Yaskawa INFORM job: u_tourne2TRJ0.JBI

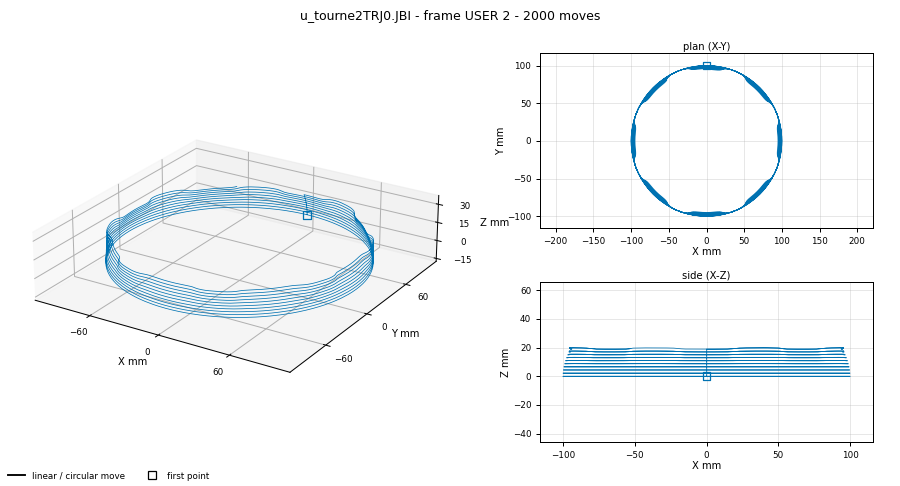
[picture p0: tool path of u_tourne2TRJ0.JBI in frame USER 2, 2000 of 2000 moves have a stored position in this frame; points joined in program order, loops and branches not executed]
/JOB
//NAME u_tourne2TRJ0
///FOLDERNAME DEMO
//POS
///NPOS 2000,0,0,0,0,0
///USER 2
///TOOL 7
///POSTYPE USER
///RECTAN
///RCONF 1,0,0,0,0,0,0,0,0,0,0,0,0,0,0,0,0,0,0,0,0,0,0,0
C00000=0.000,100.000,0.000,-180.0000,0.0000,0.0000
C00001=5.792,99.832,0.000,-180.0000,-0.0000,0.0000
C00002=10.988,99.394,0.000,-180.0000,-0.0000,0.0000
C00003=15.564,98.781,0.000,-180.0000,-0.0000,0.0000
C00004=18.698,98.237,0.000,-180.0000,-0.0000,0.0000
C00005=20.854,97.801,0.000,-180.0000,-0.0000,0.0000
C00006=22.593,97.414,0.000,-180.0000,-0.0000,0.0000
C00007=24.351,96.990,0.000,-180.0000,-0.0000,0.0000
C00008=26.550,96.411,0.000,-180.0000,-0.0000,0.0000
C00009=29.248,95.627,0.000,-180.0000,-0.0000,0.0000
C00010=32.094,94.710,0.000,-180.0000,-0.0000,0.0000
C00011=34.739,93.772,0.000,-180.0000,-0.0000,0.0000
C00012=37.121,92.855,0.000,-180.0000,-0.0000,0.0000
C00013=39.410,91.907,0.000,-180.0000,-0.0000,0.0000
C00014=41.743,90.871,0.000,-180.0000,-0.0000,0.0000
C00015=44.276,89.664,0.000,180.0000,0.0000,0.0000
C00016=46.937,88.300,0.000,180.0000,0.0000,0.0000
C00017=49.400,86.946,0.000,-180.0000,-0.0000,0.0000
C00018=51.363,85.801,0.000,-180.0000,-0.0000,0.0000
C00019=52.906,84.858,0.000,-180.0000,-0.0000,0.0000
C00020=54.410,83.902,0.000,-180.0000,-0.0000,0.0000
C00021=56.242,82.685,0.000,-180.0000,-0.0000,0.0000
C00022=58.844,80.854,0.000,-180.0000,-0.0000,0.0000
C00023=62.512,78.053,0.000,-180.0000,-0.0000,0.0000
C00024=66.496,74.687,0.000,-180.0000,-0.0000,0.0000
C00025=70.711,70.711,0.000,-180.0000,-0.0000,0.0000
C00026=74.687,66.496,0.000,-180.0000,-0.0000,0.0000
C00027=78.053,62.512,0.000,-180.0000,-0.0000,0.0000
C00028=80.854,58.844,0.000,180.0000,0.0000,0.0000
C00029=82.685,56.242,0.000,-180.0000,-0.0000,0.0000
C00030=83.902,54.410,0.000,-180.0000,-0.0000,0.0000
C00031=84.858,52.906,0.000,-180.0000,-0.0000,0.0000
C00032=85.801,51.363,0.000,-180.0000,-0.0000,0.0000
C00033=86.946,49.400,0.000,-180.0000,-0.0000,0.0000
C00034=88.300,46.937,0.000,-180.0000,-0.0000,0.0000
C00035=89.664,44.276,0.000,-180.0000,-0.0000,0.0000
C00036=90.871,41.743,0.000,-180.0000,-0.0000,0.0000
C00037=91.907,39.410,0.000,-180.0000,-0.0000,0.0000
C00038=92.855,37.121,0.000,-180.0000,-0.0000,0.0000
C00039=93.772,34.739,0.000,-180.0000,-0.0000,0.0000
C00040=94.710,32.094,0.000,-180.0000,-0.0000,0.0000
C00041=95.627,29.248,0.000,-180.0000,-0.0000,0.0000
C00042=96.411,26.550,0.000,-180.0000,-0.0000,0.0000
C00043=96.990,24.351,0.000,-180.0000,-0.0000,0.0000
C00044=97.414,22.593,0.000,-180.0000,-0.0000,0.0000
C00045=97.801,20.854,0.000,-180.0000,-0.0000,0.0000
C00046=98.237,18.698,0.000,-180.0000,-0.0000,0.0000
C00047=98.781,15.564,0.000,-180.0000,-0.0000,0.0000
C00048=99.394,10.988,0.000,-180.0000,-0.0000,0.0000
C00049=99.832,5.792,0.000,-180.0000,-0.0000,0.0000
C00050=100.000,0.000,0.000,-180.0000,-0.0000,0.0000
C00051=99.832,-5.792,0.000,180.0000,-0.0000,0.0000
C00052=99.394,-10.988,0.000,180.0000,-0.0000,0.0000
C00053=98.781,-15.564,0.000,180.0000,-0.0000,0.0000
C00054=98.237,-18.698,0.000,180.0000,-0.0000,0.0000
C00055=97.801,-20.854,0.000,180.0000,-0.0000,0.0000
C00056=97.414,-22.593,0.000,180.0000,-0.0000,0.0000
C00057=96.990,-24.351,0.000,180.0000,-0.0000,0.0000
C00058=96.411,-26.550,0.000,180.0000,-0.0000,0.0000
C00059=95.627,-29.248,0.000,180.0000,-0.0000,0.0000
C00060=94.710,-32.094,0.000,180.0000,-0.0000,0.0000
C00061=93.772,-34.739,0.000,180.0000,-0.0000,0.0000
C00062=92.855,-37.121,0.000,180.0000,-0.0000,0.0000
C00063=91.907,-39.410,0.000,180.0000,-0.0000,0.0000
C00064=90.871,-41.743,0.000,180.0000,-0.0000,0.0000
C00065=89.664,-44.276,0.000,180.0000,-0.0000,0.0000
C00066=88.300,-46.937,0.000,180.0000,-0.0000,0.0000
C00067=86.946,-49.400,0.000,180.0000,-0.0000,0.0000
C00068=85.801,-51.363,0.000,180.0000,-0.0000,0.0000
C00069=84.858,-52.906,0.000,180.0000,-0.0000,0.0000
C00070=83.902,-54.410,0.000,180.0000,-0.0000,0.0000
C00071=82.685,-56.242,0.000,180.0000,-0.0000,0.0000
C00072=80.854,-58.844,0.000,180.0000,-0.0000,0.0000
C00073=78.053,-62.512,0.000,180.0000,-0.0000,0.0000
C00074=74.687,-66.496,0.000,180.0000,-0.0000,0.0000
C00075=70.711,-70.711,0.000,180.0000,-0.0000,0.0000
C00076=66.496,-74.687,0.000,180.0000,-0.0000,0.0000
C00077=62.512,-78.053,0.000,180.0000,-0.0000,0.0000
C00078=58.844,-80.854,0.000,180.0000,-0.0000,0.0000
C00079=56.242,-82.685,0.000,180.0000,-0.0000,0.0000
C00080=54.410,-83.902,0.000,180.0000,-0.0000,0.0000
C00081=52.906,-84.858,0.000,180.0000,-0.0000,0.0000
C00082=51.363,-85.801,0.000,180.0000,-0.0000,0.0000
C00083=49.400,-86.946,0.000,-180.0000,0.0000,0.0000
C00084=46.937,-88.300,0.000,180.0000,-0.0000,0.0000
C00085=44.276,-89.664,0.000,180.0000,-0.0000,0.0000
C00086=41.743,-90.871,0.000,180.0000,-0.0000,0.0000
C00087=39.410,-91.907,0.000,180.0000,-0.0000,0.0000
C00088=37.121,-92.855,0.000,180.0000,-0.0000,0.0000
C00089=34.739,-93.772,0.000,180.0000,-0.0000,0.0000
C00090=32.094,-94.710,0.000,180.0000,-0.0000,0.0000
C00091=29.248,-95.627,0.000,180.0000,-0.0000,0.0000
C00092=26.550,-96.411,0.000,180.0000,-0.0000,0.0000
C00093=24.351,-96.990,0.000,180.0000,-0.0000,0.0000
C00094=22.593,-97.414,0.000,180.0000,-0.0000,0.0000
C00095=20.854,-97.801,0.000,180.0000,-0.0000,0.0000
C00096=18.698,-98.237,0.000,180.0000,-0.0000,0.0000
C00097=15.564,-98.781,0.000,180.0000,-0.0000,0.0000
C00098=10.988,-99.394,0.000,180.0000,-0.0000,0.0000
C00099=5.792,-99.832,0.000,180.0000,-0.0000,0.0000
C00100=0.000,-100.000,0.000,-180.0000,-0.0000,0.0000
C00101=0.000,-100.000,0.000,-180.0000,-0.0000,0.0000
C00102=-5.792,-99.832,0.000,-180.0000,-0.0000,0.0000
C00103=-10.988,-99.394,0.000,-180.0000,-0.0000,0.0000
C00104=-15.564,-98.781,0.000,-180.0000,-0.0000,0.0000
C00105=-18.698,-98.237,0.000,-180.0000,-0.0000,0.0000
C00106=-20.854,-97.801,0.000,-180.0000,-0.0000,0.0000
C00107=-22.593,-97.414,0.000,-180.0000,-0.0000,0.0000
C00108=-24.351,-96.990,0.000,-180.0000,-0.0000,0.0000
C00109=-26.550,-96.411,0.000,-180.0000,-0.0000,0.0000
C00110=-29.248,-95.627,0.000,-180.0000,-0.0000,0.0000
C00111=-32.094,-94.710,0.000,-180.0000,-0.0000,0.0000
C00112=-34.739,-93.772,0.000,-180.0000,-0.0000,0.0000
C00113=-37.121,-92.855,0.000,-180.0000,-0.0000,0.0000
C00114=-39.410,-91.907,0.000,-180.0000,-0.0000,0.0000
C00115=-41.743,-90.871,0.000,-180.0000,-0.0000,0.0000
C00116=-44.276,-89.664,0.000,-180.0000,-0.0000,0.0000
C00117=-46.937,-88.300,0.000,-180.0000,-0.0000,0.0000
C00118=-49.400,-86.946,0.000,-180.0000,-0.0000,0.0000
C00119=-51.363,-85.801,0.000,-180.0000,-0.0000,0.0000
C00120=-52.906,-84.858,0.000,-180.0000,-0.0000,0.0000
C00121=-54.410,-83.902,0.000,-180.0000,-0.0000,0.0000
C00122=-56.242,-82.685,0.000,-180.0000,-0.0000,0.0000
C00123=-58.844,-80.854,0.000,-180.0000,-0.0000,0.0000
C00124=-62.512,-78.053,0.000,-180.0000,-0.0000,0.0000
C00125=-66.496,-74.687,0.000,-180.0000,-0.0000,0.0000
C00126=-70.711,-70.711,0.000,-180.0000,-0.0000,0.0000
C00127=-74.687,-66.496,0.000,-180.0000,-0.0000,0.0000
C00128=-78.053,-62.512,0.000,-180.0000,-0.0000,0.0000
C00129=-80.854,-58.844,0.000,-180.0000,-0.0000,0.0000
C00130=-82.685,-56.242,0.000,-180.0000,-0.0000,0.0000
C00131=-83.902,-54.410,0.000,-180.0000,-0.0000,0.0000
C00132=-84.858,-52.906,0.000,-180.0000,-0.0000,0.0000
C00133=-85.801,-51.363,0.000,-180.0000,-0.0000,0.0000
C00134=-86.946,-49.400,0.000,-180.0000,-0.0000,0.0000
C00135=-88.300,-46.937,0.000,-180.0000,-0.0000,0.0000
C00136=-89.664,-44.276,0.000,-180.0000,-0.0000,0.0000
C00137=-90.871,-41.743,0.000,180.0000,0.0000,0.0000
C00138=-91.907,-39.410,0.000,180.0000,0.0000,0.0000
C00139=-92.855,-37.121,0.000,-180.0000,-0.0000,0.0000
C00140=-93.772,-34.739,0.000,-180.0000,-0.0000,0.0000
C00141=-94.710,-32.094,0.000,180.0000,0.0000,0.0000
C00142=-95.627,-29.248,0.000,180.0000,0.0000,0.0000
C00143=-96.411,-26.550,0.000,-180.0000,-0.0000,0.0000
C00144=-96.990,-24.351,0.000,-180.0000,-0.0000,0.0000
C00145=-97.414,-22.593,0.000,-180.0000,-0.0000,0.0000
C00146=-97.801,-20.854,0.000,-180.0000,-0.0000,0.0000
C00147=-98.237,-18.698,0.000,-180.0000,-0.0000,0.0000
C00148=-98.781,-15.564,0.000,-180.0000,-0.0000,0.0000
C00149=-99.394,-10.988,0.000,-180.0000,-0.0000,0.0000
C00150=-99.832,-5.792,0.000,-180.0000,-0.0000,0.0000
C00151=-100.000,0.000,0.000,180.0000,0.0000,0.0000
C00152=-99.832,5.792,0.000,-180.0000,0.0000,0.0000
C00153=-99.394,10.988,0.000,-180.0000,0.0000,0.0000
C00154=-98.781,15.564,0.000,-180.0000,0.0000,0.0000
C00155=-98.237,18.698,0.000,-180.0000,0.0000,0.0000
C00156=-97.801,20.854,0.000,-180.0000,0.0000,0.0000
C00157=-97.414,22.593,0.000,-180.0000,0.0000,0.0000
C00158=-96.990,24.351,0.000,-180.0000,0.0000,0.0000
C00159=-96.411,26.550,0.000,-180.0000,0.0000,0.0000
C00160=-95.627,29.248,0.000,-180.0000,0.0000,0.0000
C00161=-94.710,32.094,0.000,-180.0000,0.0000,0.0000
C00162=-93.772,34.739,0.000,-180.0000,0.0000,0.0000
C00163=-92.855,37.121,0.000,-180.0000,0.0000,0.0000
C00164=-91.907,39.410,0.000,-180.0000,0.0000,0.0000
C00165=-90.871,41.743,0.000,-180.0000,0.0000,0.0000
C00166=-89.664,44.276,0.000,-180.0000,0.0000,0.0000
C00167=-88.300,46.937,0.000,-180.0000,0.0000,0.0000
C00168=-86.946,49.400,0.000,-180.0000,0.0000,0.0000
C00169=-85.801,51.363,0.000,-180.0000,0.0000,0.0000
C00170=-84.858,52.906,0.000,-180.0000,0.0000,0.0000
C00171=-83.902,54.410,0.000,-180.0000,0.0000,0.0000
C00172=-82.685,56.242,0.000,-180.0000,0.0000,0.0000
C00173=-80.854,58.844,0.000,-180.0000,0.0000,0.0000
C00174=-78.053,62.512,0.000,-180.0000,0.0000,0.0000
C00175=-74.687,66.496,0.000,-180.0000,0.0000,0.0000
C00176=-70.711,70.711,0.000,-180.0000,0.0000,0.0000
C00177=-66.496,74.687,0.000,-180.0000,0.0000,0.0000
C00178=-62.512,78.053,0.000,-180.0000,0.0000,0.0000
C00179=-58.844,80.854,0.000,-180.0000,0.0000,0.0000
C00180=-56.242,82.685,0.000,-180.0000,0.0000,0.0000
C00181=-54.410,83.902,0.000,-180.0000,0.0000,0.0000
C00182=-52.906,84.858,0.000,-180.0000,0.0000,0.0000
C00183=-51.363,85.801,0.000,-180.0000,0.0000,0.0000
C00184=-49.400,86.946,0.000,-180.0000,0.0000,0.0000
C00185=-46.937,88.300,0.000,-180.0000,0.0000,0.0000
C00186=-44.276,89.664,0.000,-180.0000,0.0000,0.0000
C00187=-41.743,90.871,0.000,-180.0000,0.0000,0.0000
C00188=-39.410,91.907,0.000,-180.0000,0.0000,0.0000
C00189=-37.121,92.855,0.000,-180.0000,0.0000,0.0000
C00190=-34.739,93.772,0.000,-180.0000,0.0000,0.0000
C00191=-32.094,94.710,0.000,-180.0000,0.0000,0.0000
C00192=-29.248,95.627,0.000,-180.0000,0.0000,0.0000
C00193=-26.550,96.411,0.000,-180.0000,0.0000,0.0000
C00194=-24.351,96.990,0.000,-180.0000,0.0000,0.0000
C00195=-22.593,97.414,0.000,-180.0000,0.0000,0.0000
C00196=-20.854,97.801,0.000,-180.0000,0.0000,0.0000
C00197=-18.698,98.237,0.000,-180.0000,0.0000,0.0000
C00198=-15.564,98.781,0.000,-180.0000,0.0000,0.0000
C00199=-10.988,99.394,0.000,-180.0000,0.0000,0.0000
C00200=-5.792,99.832,0.000,-180.0000,0.0000,0.0000
C00201=0.000,100.000,0.000,-180.0000,0.0000,0.0000
C00202=0.000,99.921,2.199,-175.9401,0.0000,0.0000
C00203=5.785,99.754,2.199,-175.9458,-0.2355,0.0000
C00204=10.976,99.317,2.199,-175.9687,-0.4480,0.0000
C00205=15.549,98.707,2.199,-176.1467,-0.6030,0.0000
C00206=18.681,98.171,2.199,-176.5598,-0.6429,0.0000
C00207=20.835,97.748,2.199,-177.1510,-0.5909,0.0000
C00208=22.573,97.375,2.200,-177.8335,-0.4817,0.0000
C00209=24.330,96.965,2.200,-178.5158,-0.3611,0.0000
C00210=26.527,96.399,2.200,-179.1062,-0.2407,0.0000
C00211=29.226,95.625,2.200,-179.5703,-0.1318,0.0000
C00212=32.077,94.713,2.200,-179.8797,-0.0401,0.0000
C00213=34.728,93.776,2.200,-179.9828,-0.0057,0.0000
C00214=37.118,92.856,2.200,-180.0000,-0.0000,0.0000
C00215=39.413,91.905,2.200,-180.0000,-0.0000,0.0000
C00216=41.753,90.866,2.200,-179.9828,-0.0115,0.0000
C00217=44.291,89.654,2.200,-179.8854,-0.0573,0.0000
C00218=46.951,88.283,2.200,-179.6047,-0.2120,0.0000
C00219=49.407,86.922,2.200,-179.1978,-0.4641,0.0000
C00220=51.360,85.768,2.200,-178.6934,-0.7909,0.0000
C00221=52.893,84.816,2.200,-178.1256,-1.1925,0.0000
C00222=54.385,83.851,2.199,-177.5690,-1.6002,0.0000
C00223=56.208,82.627,2.199,-177.1150,-1.9797,0.0000
C00224=58.802,80.791,2.199,-176.8504,-2.3016,0.0000
C00225=62.466,77.989,2.199,-176.8326,-2.5372,0.0000
C00226=66.446,74.627,2.199,-176.9643,-2.7034,0.0000
C00227=70.655,70.655,2.199,-177.1247,-2.8753,0.0000
C00228=74.627,66.446,2.199,-177.2966,-3.0357,0.0000
C00229=77.989,62.466,2.199,-177.4628,-3.1674,0.0000
C00230=80.791,58.802,2.199,-177.6984,-3.1496,0.0000
C00231=82.627,56.208,2.199,-178.0203,-2.8850,0.0000
C00232=83.851,54.385,2.199,-178.3998,-2.4310,0.0000
C00233=84.816,52.893,2.200,-178.8075,-1.8744,0.0000
C00234=85.768,51.360,2.200,-179.2091,-1.3066,0.0000
C00235=86.922,49.407,2.200,-179.5359,-0.8022,0.0000
C00236=88.283,46.951,2.200,-179.7880,-0.3953,0.0000
C00237=89.654,44.291,2.200,-179.9427,-0.1146,0.0000
C00238=90.866,41.753,2.200,-179.9885,-0.0172,0.0000
C00239=91.905,39.413,2.200,-180.0000,-0.0000,0.0000
C00240=92.856,37.118,2.200,-180.0000,-0.0000,0.0000
C00241=93.776,34.728,2.200,-179.9943,-0.0172,0.0000
C00242=94.713,32.077,2.200,-179.9599,-0.1203,0.0000
C00243=95.625,29.226,2.200,-179.8682,-0.4297,0.0000
C00244=96.399,26.527,2.200,-179.7593,-0.8938,0.0000
C00245=96.965,24.330,2.200,-179.6389,-1.4842,0.0000
C00246=97.375,22.573,2.200,-179.5183,-2.1665,0.0000
C00247=97.748,20.835,2.199,-179.4091,-2.8490,0.0000
C00248=98.171,18.681,2.199,-179.3571,-3.4402,0.0000
C00249=98.707,15.549,2.199,-179.3970,-3.8533,0.0000
C00250=99.317,10.976,2.199,-179.5520,-4.0313,0.0000
C00251=99.754,5.785,2.199,-179.7645,-4.0542,0.0000
C00252=99.921,0.000,2.199,180.0000,-4.0599,0.0000
C00253=99.754,-5.785,2.199,179.7645,-4.0542,0.0000
C00254=99.317,-10.976,2.199,179.5520,-4.0313,0.0000
C00255=98.707,-15.549,2.199,179.3970,-3.8533,0.0000
C00256=98.171,-18.681,2.199,179.3571,-3.4402,0.0000
C00257=97.748,-20.835,2.199,179.4091,-2.8490,0.0000
C00258=97.375,-22.573,2.200,179.5183,-2.1665,0.0000
C00259=96.965,-24.330,2.200,179.6389,-1.4842,0.0000
C00260=96.399,-26.527,2.200,179.7593,-0.8938,0.0000
C00261=95.625,-29.226,2.200,179.8682,-0.4297,0.0000
C00262=94.713,-32.077,2.200,179.9599,-0.1203,0.0000
C00263=93.776,-34.728,2.200,179.9943,-0.0172,0.0000
C00264=92.856,-37.118,2.200,180.0000,-0.0000,0.0000
C00265=91.905,-39.413,2.200,180.0000,-0.0000,0.0000
C00266=90.866,-41.753,2.200,179.9885,-0.0172,0.0000
C00267=89.654,-44.291,2.200,179.9427,-0.1146,0.0000
C00268=88.283,-46.951,2.200,179.7880,-0.3953,0.0000
C00269=86.922,-49.407,2.200,179.5359,-0.8022,0.0000
C00270=85.768,-51.360,2.200,179.2091,-1.3066,0.0000
C00271=84.816,-52.893,2.200,178.8075,-1.8744,0.0000
C00272=83.851,-54.385,2.199,178.3998,-2.4310,0.0000
C00273=82.627,-56.208,2.199,178.0203,-2.8850,0.0000
C00274=80.791,-58.802,2.199,177.6984,-3.1496,0.0000
C00275=77.989,-62.466,2.199,177.4628,-3.1674,0.0000
C00276=74.627,-66.446,2.199,177.2966,-3.0357,0.0000
C00277=70.655,-70.655,2.199,177.1247,-2.8753,0.0000
C00278=66.446,-74.627,2.199,176.9643,-2.7034,0.0000
C00279=62.466,-77.989,2.199,176.8326,-2.5372,0.0000
C00280=58.802,-80.791,2.199,176.8504,-2.3016,0.0000
C00281=56.208,-82.627,2.199,177.1150,-1.9797,0.0000
C00282=54.385,-83.851,2.199,177.5690,-1.6002,0.0000
C00283=52.893,-84.816,2.200,178.1256,-1.1925,0.0000
C00284=51.360,-85.768,2.200,178.6934,-0.7909,0.0000
C00285=49.407,-86.922,2.200,179.1978,-0.4641,0.0000
C00286=46.951,-88.283,2.200,179.6047,-0.2120,0.0000
C00287=44.291,-89.654,2.200,179.8854,-0.0573,0.0000
C00288=41.753,-90.866,2.200,179.9828,-0.0115,0.0000
C00289=39.413,-91.905,2.200,180.0000,-0.0000,0.0000
C00290=37.118,-92.856,2.200,180.0000,-0.0000,0.0000
C00291=34.728,-93.776,2.200,179.9828,-0.0057,0.0000
C00292=32.077,-94.713,2.200,179.8797,-0.0401,0.0000
C00293=29.226,-95.625,2.200,179.5703,-0.1318,0.0000
C00294=26.527,-96.399,2.200,179.1062,-0.2407,0.0000
C00295=24.330,-96.965,2.200,178.5158,-0.3611,0.0000
C00296=22.573,-97.375,2.200,177.8335,-0.4817,0.0000
C00297=20.835,-97.748,2.199,177.1510,-0.5909,0.0000
C00298=18.681,-98.171,2.199,176.5598,-0.6429,0.0000
C00299=15.549,-98.707,2.199,176.1467,-0.6030,0.0000
C00300=10.976,-99.317,2.199,175.9687,-0.4480,0.0000
C00301=5.785,-99.754,2.199,175.9458,-0.2355,0.0000
C00302=0.000,-99.921,2.199,175.9401,0.0000,0.0000
C00303=0.000,-99.921,2.199,175.9401,0.0000,0.0000
C00304=-5.785,-99.754,2.199,175.9458,0.2355,0.0000
C00305=-10.976,-99.317,2.199,175.9687,0.4480,0.0000
C00306=-15.549,-98.707,2.199,176.1467,0.6030,0.0000
C00307=-18.681,-98.171,2.199,176.5598,0.6429,0.0000
C00308=-20.835,-97.748,2.199,177.1510,0.5909,0.0000
C00309=-22.573,-97.375,2.200,177.8335,0.4817,0.0000
C00310=-24.330,-96.965,2.200,178.5158,0.3611,0.0000
C00311=-26.527,-96.399,2.200,179.1062,0.2407,0.0000
C00312=-29.226,-95.625,2.200,179.5703,0.1318,0.0000
C00313=-32.077,-94.713,2.200,179.8797,0.0401,0.0000
C00314=-34.728,-93.776,2.200,179.9828,0.0057,0.0000
C00315=-37.118,-92.856,2.200,180.0000,0.0000,0.0000
C00316=-39.413,-91.905,2.200,180.0000,0.0000,0.0000
C00317=-41.753,-90.866,2.200,179.9828,0.0115,0.0000
C00318=-44.291,-89.654,2.200,179.8854,0.0573,0.0000
C00319=-46.951,-88.283,2.200,179.6047,0.2120,0.0000
C00320=-49.407,-86.922,2.200,179.1978,0.4641,0.0000
C00321=-51.360,-85.768,2.200,178.6934,0.7909,0.0000
C00322=-52.893,-84.816,2.200,178.1256,1.1925,0.0000
C00323=-54.385,-83.851,2.199,177.5690,1.6002,0.0000
C00324=-56.208,-82.627,2.199,177.1150,1.9797,0.0000
C00325=-58.802,-80.791,2.199,176.8504,2.3016,0.0000
C00326=-62.466,-77.989,2.199,176.8326,2.5372,0.0000
C00327=-66.446,-74.627,2.199,176.9643,2.7034,0.0000
C00328=-70.655,-70.655,2.199,177.1247,2.8753,0.0000
C00329=-74.627,-66.446,2.199,177.2966,3.0357,0.0000
C00330=-77.989,-62.466,2.199,177.4628,3.1674,0.0000
C00331=-80.791,-58.802,2.199,177.6984,3.1496,0.0000
C00332=-82.627,-56.208,2.199,178.0203,2.8850,0.0000
C00333=-83.851,-54.385,2.199,178.3998,2.4310,0.0000
C00334=-84.816,-52.893,2.200,178.8075,1.8744,0.0000
C00335=-85.768,-51.360,2.200,179.2091,1.3066,0.0000
C00336=-86.922,-49.407,2.200,179.5359,0.8022,0.0000
C00337=-88.283,-46.951,2.200,179.7880,0.3953,0.0000
C00338=-89.654,-44.291,2.200,179.9427,0.1146,0.0000
C00339=-90.866,-41.753,2.200,179.9885,0.0172,0.0000
C00340=-91.905,-39.413,2.200,180.0000,0.0000,0.0000
C00341=-92.856,-37.118,2.200,180.0000,0.0000,0.0000
C00342=-93.776,-34.728,2.200,179.9943,0.0172,0.0000
C00343=-94.713,-32.077,2.200,179.9599,0.1203,0.0000
C00344=-95.625,-29.226,2.200,179.8682,0.4297,0.0000
C00345=-96.399,-26.527,2.200,179.7593,0.8938,0.0000
C00346=-96.965,-24.330,2.200,179.6389,1.4842,0.0000
C00347=-97.375,-22.573,2.200,179.5183,2.1665,0.0000
C00348=-97.748,-20.835,2.199,179.4091,2.8490,0.0000
C00349=-98.171,-18.681,2.199,179.3571,3.4402,0.0000
C00350=-98.707,-15.549,2.199,179.3970,3.8533,0.0000
C00351=-99.317,-10.976,2.199,179.5520,4.0313,0.0000
C00352=-99.754,-5.785,2.199,179.7645,4.0542,0.0000
C00353=-99.921,0.000,2.199,-180.0000,4.0599,0.0000
C00354=-99.754,5.785,2.199,-179.7645,4.0542,0.0000
C00355=-99.317,10.976,2.199,-179.5520,4.0313,0.0000
C00356=-98.707,15.549,2.199,-179.3970,3.8533,0.0000
C00357=-98.171,18.681,2.199,-179.3571,3.4402,0.0000
C00358=-97.748,20.835,2.199,-179.4091,2.8490,0.0000
C00359=-97.375,22.573,2.200,-179.5183,2.1665,0.0000
C00360=-96.965,24.330,2.200,-179.6389,1.4842,0.0000
C00361=-96.399,26.527,2.200,-179.7593,0.8938,0.0000
C00362=-95.625,29.226,2.200,-179.8682,0.4297,0.0000
C00363=-94.713,32.077,2.200,-179.9599,0.1203,0.0000
C00364=-93.776,34.728,2.200,-179.9943,0.0172,0.0000
C00365=-92.856,37.118,2.200,-180.0000,0.0000,0.0000
C00366=-91.905,39.413,2.200,-180.0000,0.0000,0.0000
C00367=-90.866,41.753,2.200,-179.9885,0.0172,0.0000
C00368=-89.654,44.291,2.200,-179.9427,0.1146,0.0000
C00369=-88.283,46.951,2.200,-179.7880,0.3953,0.0000
C00370=-86.922,49.407,2.200,-179.5359,0.8022,0.0000
C00371=-85.768,51.360,2.200,-179.2091,1.3066,0.0000
C00372=-84.816,52.893,2.200,-178.8075,1.8744,0.0000
C00373=-83.851,54.385,2.199,-178.3998,2.4310,0.0000
C00374=-82.627,56.208,2.199,-178.0203,2.8850,0.0000
C00375=-80.791,58.802,2.199,-177.6984,3.1496,0.0000
C00376=-77.989,62.466,2.199,-177.4628,3.1674,0.0000
C00377=-74.627,66.446,2.199,-177.2966,3.0357,0.0000
C00378=-70.655,70.655,2.199,-177.1247,2.8753,0.0000
C00379=-66.446,74.627,2.199,-176.9643,2.7034,0.0000
C00380=-62.466,77.989,2.199,-176.8326,2.5372,0.0000
C00381=-58.802,80.791,2.199,-176.8504,2.3016,0.0000
C00382=-56.208,82.627,2.199,-177.1150,1.9797,0.0000
C00383=-54.385,83.851,2.199,-177.5690,1.6002,0.0000
C00384=-52.893,84.816,2.200,-178.1256,1.1925,0.0000
C00385=-51.360,85.768,2.200,-178.6934,0.7909,0.0000
C00386=-49.407,86.922,2.200,-179.1978,0.4641,0.0000
C00387=-46.951,88.283,2.200,-179.6047,0.2120,0.0000
C00388=-44.291,89.654,2.200,-179.8854,0.0573,0.0000
C00389=-41.753,90.866,2.200,-179.9828,0.0115,0.0000
C00390=-39.413,91.905,2.200,-180.0000,0.0000,0.0000
C00391=-37.118,92.856,2.200,-180.0000,0.0000,0.0000
C00392=-34.728,93.776,2.200,-179.9828,0.0057,0.0000
C00393=-32.077,94.713,2.200,-179.8797,0.0401,0.0000
C00394=-29.226,95.625,2.200,-179.5703,0.1318,0.0000
C00395=-26.527,96.399,2.200,-179.1062,0.2407,0.0000
C00396=-24.330,96.965,2.200,-178.5158,0.3611,0.0000
C00397=-22.573,97.375,2.200,-177.8335,0.4817,0.0000
C00398=-20.835,97.748,2.199,-177.1510,0.5909,0.0000
C00399=-18.681,98.171,2.199,-176.5598,0.6429,0.0000
C00400=-15.549,98.707,2.199,-176.1467,0.6030,0.0000
C00401=-10.976,99.317,2.199,-175.9687,0.4480,0.0000
C00402=-5.785,99.754,2.199,-175.9458,0.2355,0.0000
C00403=0.000,99.921,2.199,-175.9401,0.0000,0.0000
C00404=0.000,99.691,4.387,-172.1025,0.0000,0.0000
C00405=5.764,99.524,4.387,-172.1138,-0.4628,0.0000
C00406=10.941,99.090,4.387,-172.1592,-0.8618,0.0000
C00407=15.506,98.490,4.388,-172.4997,-1.1444,0.0000
C00408=18.630,97.979,4.390,-173.2915,-1.1769,0.0000
C00409=20.779,97.591,4.393,-174.4382,-1.0363,0.0000
C00410=22.514,97.259,4.396,-175.7731,-0.8388,0.0000
C00411=24.268,96.890,4.398,-177.1167,-0.6425,0.0000
C00412=26.460,96.362,4.399,-178.2693,-0.4471,0.0000
C00413=29.164,95.617,4.399,-179.1806,-0.2407,0.0000
C00414=32.027,94.722,4.399,-179.7708,-0.0745,0.0000
C00415=34.697,93.786,4.400,-179.9656,-0.0115,0.0000
C00416=37.107,92.860,4.400,-179.9943,-0.0000,0.0000
C00417=39.424,91.901,4.400,-179.9943,-0.0000,0.0000
C00418=41.782,90.851,4.400,-179.9656,-0.0172,0.0000
C00419=44.332,89.625,4.399,-179.7823,-0.1089,0.0000
C00420=46.990,88.233,4.399,-179.2494,-0.4126,0.0000
C00421=49.428,86.848,4.399,-178.4583,-0.9114,0.0000
C00422=51.352,85.672,4.398,-177.5060,-1.5830,0.0000
C00423=52.853,84.692,4.396,-176.4194,-2.4003,0.0000
C00424=54.314,83.700,4.393,-175.3293,-3.2095,0.0000
C00425=56.108,82.455,4.390,-174.4208,-3.9289,0.0000
C00426=58.679,80.608,4.388,-173.8788,-4.5167,0.0000
C00427=62.331,77.804,4.387,-173.8345,-4.9565,0.0000
C00428=66.299,74.450,4.387,-174.0804,-5.2721,0.0000
C00429=70.493,70.493,4.387,-174.3954,-5.6046,0.0000
C00430=74.450,66.299,4.387,-174.7279,-5.9196,0.0000
C00431=77.804,62.331,4.387,-175.0435,-6.1655,0.0000
C00432=80.608,58.679,4.388,-175.4833,-6.1212,0.0000
C00433=82.455,56.108,4.390,-176.0711,-5.5792,0.0000
C00434=83.700,54.314,4.393,-176.7905,-4.6707,0.0000
C00435=84.692,52.853,4.396,-177.5997,-3.5806,0.0000
C00436=85.672,51.352,4.398,-178.4170,-2.4940,0.0000
C00437=86.848,49.428,4.399,-179.0886,-1.5417,0.0000
C00438=88.233,46.990,4.399,-179.5874,-0.7506,0.0000
C00439=89.625,44.332,4.399,-179.8911,-0.2177,0.0000
C00440=90.851,41.782,4.400,-179.9828,-0.0344,0.0000
C00441=91.901,39.424,4.400,-180.0000,-0.0057,0.0000
C00442=92.860,37.107,4.400,-180.0000,-0.0057,0.0000
C00443=93.786,34.697,4.400,-179.9885,-0.0344,0.0000
C00444=94.722,32.027,4.399,-179.9255,-0.2292,0.0000
C00445=95.617,29.164,4.399,-179.7593,-0.8194,0.0000
C00446=96.362,26.460,4.399,-179.5529,-1.7307,0.0000
C00447=96.890,24.268,4.398,-179.3575,-2.8833,0.0000
C00448=97.259,22.514,4.396,-179.1612,-4.2269,0.0000
C00449=97.591,20.779,4.393,-178.9637,-5.5618,0.0000
C00450=97.979,18.630,4.390,-178.8231,-6.7085,0.0000
C00451=98.490,15.506,4.388,-178.8556,-7.5003,0.0000
C00452=99.090,10.941,4.387,-179.1382,-7.8408,0.0000
C00453=99.524,5.764,4.387,-179.5372,-7.8862,0.0000
C00454=99.691,0.000,4.387,180.0000,-7.8975,0.0000
C00455=99.524,-5.764,4.387,179.5372,-7.8862,0.0000
C00456=99.090,-10.941,4.387,179.1382,-7.8408,0.0000
C00457=98.490,-15.506,4.388,178.8556,-7.5003,0.0000
C00458=97.979,-18.630,4.390,178.8231,-6.7085,0.0000
C00459=97.591,-20.779,4.393,178.9637,-5.5618,0.0000
C00460=97.259,-22.514,4.396,179.1612,-4.2269,0.0000
C00461=96.890,-24.268,4.398,179.3575,-2.8833,0.0000
C00462=96.362,-26.460,4.399,179.5529,-1.7307,0.0000
C00463=95.617,-29.164,4.399,179.7593,-0.8194,0.0000
C00464=94.722,-32.027,4.399,179.9255,-0.2292,0.0000
C00465=93.786,-34.697,4.400,179.9885,-0.0344,0.0000
C00466=92.860,-37.107,4.400,180.0000,-0.0057,0.0000
C00467=91.901,-39.424,4.400,180.0000,-0.0057,0.0000
C00468=90.851,-41.782,4.400,179.9828,-0.0344,0.0000
C00469=89.625,-44.332,4.399,179.8911,-0.2177,0.0000
C00470=88.233,-46.990,4.399,179.5874,-0.7506,0.0000
C00471=86.848,-49.428,4.399,179.0886,-1.5417,0.0000
C00472=85.672,-51.352,4.398,178.4170,-2.4940,0.0000
C00473=84.692,-52.853,4.396,177.5997,-3.5806,0.0000
C00474=83.700,-54.314,4.393,176.7905,-4.6707,0.0000
C00475=82.455,-56.108,4.390,176.0711,-5.5792,0.0000
C00476=80.608,-58.679,4.388,175.4833,-6.1212,0.0000
C00477=77.804,-62.331,4.387,175.0435,-6.1655,0.0000
C00478=74.450,-66.299,4.387,174.7279,-5.9196,0.0000
C00479=70.493,-70.493,4.387,174.3954,-5.6046,0.0000
C00480=66.299,-74.450,4.387,174.0804,-5.2721,0.0000
C00481=62.331,-77.804,4.387,173.8345,-4.9565,0.0000
C00482=58.679,-80.608,4.388,173.8788,-4.5167,0.0000
C00483=56.108,-82.455,4.390,174.4208,-3.9289,0.0000
C00484=54.314,-83.700,4.393,175.3293,-3.2095,0.0000
C00485=52.853,-84.692,4.396,176.4194,-2.4003,0.0000
C00486=51.352,-85.672,4.398,177.5060,-1.5830,0.0000
C00487=49.428,-86.848,4.399,178.4583,-0.9114,0.0000
C00488=46.990,-88.233,4.399,179.2494,-0.4126,0.0000
C00489=44.332,-89.625,4.399,179.7823,-0.1089,0.0000
C00490=41.782,-90.851,4.400,179.9656,-0.0172,0.0000
C00491=39.424,-91.901,4.400,179.9943,-0.0000,0.0000
C00492=37.107,-92.860,4.400,179.9943,-0.0000,0.0000
C00493=34.697,-93.786,4.400,179.9656,-0.0115,0.0000
C00494=32.027,-94.722,4.399,179.7708,-0.0745,0.0000
C00495=29.164,-95.617,4.399,179.1806,-0.2407,0.0000
C00496=26.460,-96.362,4.399,178.2693,-0.4471,0.0000
C00497=24.268,-96.890,4.398,177.1167,-0.6425,0.0000
C00498=22.514,-97.259,4.396,175.7731,-0.8388,0.0000
C00499=20.779,-97.591,4.393,174.4382,-1.0363,0.0000
C00500=18.630,-97.979,4.390,173.2915,-1.1769,0.0000
C00501=15.506,-98.490,4.388,172.4997,-1.1444,0.0000
C00502=10.941,-99.090,4.387,172.1592,-0.8618,0.0000
C00503=5.764,-99.524,4.387,172.1138,-0.4628,0.0000
C00504=0.000,-99.691,4.387,172.1025,0.0000,0.0000
C00505=0.000,-99.691,4.387,172.1025,0.0000,0.0000
C00506=-5.764,-99.524,4.387,172.1138,0.4628,0.0000
C00507=-10.941,-99.090,4.387,172.1592,0.8618,0.0000
C00508=-15.506,-98.490,4.388,172.4997,1.1444,0.0000
C00509=-18.630,-97.979,4.390,173.2915,1.1769,0.0000
C00510=-20.779,-97.591,4.393,174.4382,1.0363,0.0000
C00511=-22.514,-97.259,4.396,175.7731,0.8388,0.0000
C00512=-24.268,-96.890,4.398,177.1167,0.6425,0.0000
C00513=-26.460,-96.362,4.399,178.2693,0.4471,0.0000
C00514=-29.164,-95.617,4.399,179.1806,0.2407,0.0000
C00515=-32.027,-94.722,4.399,179.7708,0.0745,0.0000
C00516=-34.697,-93.786,4.400,179.9656,0.0115,0.0000
C00517=-37.107,-92.860,4.400,179.9943,0.0000,0.0000
C00518=-39.424,-91.901,4.400,179.9943,0.0000,0.0000
C00519=-41.782,-90.851,4.400,179.9656,0.0172,0.0000
C00520=-44.332,-89.625,4.399,179.7823,0.1089,0.0000
C00521=-46.990,-88.233,4.399,179.2494,0.4126,0.0000
C00522=-49.428,-86.848,4.399,178.4583,0.9114,0.0000
C00523=-51.352,-85.672,4.398,177.5060,1.5830,0.0000
C00524=-52.853,-84.692,4.396,176.4194,2.4003,0.0000
C00525=-54.314,-83.700,4.393,175.3293,3.2095,0.0000
C00526=-56.108,-82.455,4.390,174.4208,3.9289,0.0000
C00527=-58.679,-80.608,4.388,173.8788,4.5167,0.0000
C00528=-62.331,-77.804,4.387,173.8345,4.9565,0.0000
C00529=-66.299,-74.450,4.387,174.0804,5.2721,0.0000
C00530=-70.493,-70.493,4.387,174.3954,5.6046,0.0000
C00531=-74.450,-66.299,4.387,174.7279,5.9196,0.0000
C00532=-77.804,-62.331,4.387,175.0435,6.1655,0.0000
C00533=-80.608,-58.679,4.388,175.4833,6.1212,0.0000
C00534=-82.455,-56.108,4.390,176.0711,5.5792,0.0000
C00535=-83.700,-54.314,4.393,176.7905,4.6707,0.0000
C00536=-84.692,-52.853,4.396,177.5997,3.5806,0.0000
C00537=-85.672,-51.352,4.398,178.4170,2.4940,0.0000
C00538=-86.848,-49.428,4.399,179.0886,1.5417,0.0000
C00539=-88.233,-46.990,4.399,179.5874,0.7506,0.0000
C00540=-89.625,-44.332,4.399,179.8911,0.2177,0.0000
C00541=-90.851,-41.782,4.400,179.9828,0.0344,0.0000
C00542=-91.901,-39.424,4.400,180.0000,0.0057,0.0000
C00543=-92.860,-37.107,4.400,180.0000,0.0057,0.0000
C00544=-93.786,-34.697,4.400,179.9885,0.0344,0.0000
C00545=-94.722,-32.027,4.399,179.9255,0.2292,0.0000
C00546=-95.617,-29.164,4.399,179.7593,0.8194,0.0000
C00547=-96.362,-26.460,4.399,179.5529,1.7307,0.0000
C00548=-96.890,-24.268,4.398,179.3575,2.8833,0.0000
C00549=-97.259,-22.514,4.396,179.1612,4.2269,0.0000
C00550=-97.591,-20.779,4.393,178.9637,5.5618,0.0000
C00551=-97.979,-18.630,4.390,178.8231,6.7085,0.0000
C00552=-98.490,-15.506,4.388,178.8556,7.5003,0.0000
C00553=-99.090,-10.941,4.387,179.1382,7.8408,0.0000
C00554=-99.524,-5.764,4.387,179.5372,7.8862,0.0000
C00555=-99.691,0.000,4.387,-180.0000,7.8975,0.0000
C00556=-99.524,5.764,4.387,-179.5372,7.8862,0.0000
C00557=-99.090,10.941,4.387,-179.1382,7.8408,0.0000
C00558=-98.490,15.506,4.388,-178.8556,7.5003,0.0000
C00559=-97.979,18.630,4.390,-178.8231,6.7085,0.0000
C00560=-97.591,20.779,4.393,-178.9637,5.5618,0.0000
C00561=-97.259,22.514,4.396,-179.1612,4.2269,0.0000
C00562=-96.890,24.268,4.398,-179.3575,2.8833,0.0000
C00563=-96.362,26.460,4.399,-179.5529,1.7307,0.0000
C00564=-95.617,29.164,4.399,-179.7593,0.8194,0.0000
C00565=-94.722,32.027,4.399,-179.9255,0.2292,0.0000
C00566=-93.786,34.697,4.400,-179.9885,0.0344,0.0000
C00567=-92.860,37.107,4.400,-180.0000,0.0057,0.0000
C00568=-91.901,39.424,4.400,-180.0000,0.0057,0.0000
C00569=-90.851,41.782,4.400,-179.9828,0.0344,0.0000
C00570=-89.625,44.332,4.399,-179.8911,0.2177,0.0000
C00571=-88.233,46.990,4.399,-179.5874,0.7506,0.0000
C00572=-86.848,49.428,4.399,-179.0886,1.5417,0.0000
C00573=-85.672,51.352,4.398,-178.4170,2.4940,0.0000
C00574=-84.692,52.853,4.396,-177.5997,3.5806,0.0000
C00575=-83.700,54.314,4.393,-176.7905,4.6707,0.0000
C00576=-82.455,56.108,4.390,-176.0711,5.5792,0.0000
C00577=-80.608,58.679,4.388,-175.4833,6.1212,0.0000
C00578=-77.804,62.331,4.387,-175.0435,6.1655,0.0000
C00579=-74.450,66.299,4.387,-174.7279,5.9196,0.0000
C00580=-70.493,70.493,4.387,-174.3954,5.6046,0.0000
C00581=-66.299,74.450,4.387,-174.0804,5.2721,0.0000
C00582=-62.331,77.804,4.387,-173.8345,4.9565,0.0000
C00583=-58.679,80.608,4.388,-173.8788,4.5167,0.0000
C00584=-56.108,82.455,4.390,-174.4208,3.9289,0.0000
C00585=-54.314,83.700,4.393,-175.3293,3.2095,0.0000
C00586=-52.853,84.692,4.396,-176.4194,2.4003,0.0000
C00587=-51.352,85.672,4.398,-177.5060,1.5830,0.0000
C00588=-49.428,86.848,4.399,-178.4583,0.9114,0.0000
C00589=-46.990,88.233,4.399,-179.2494,0.4126,0.0000
C00590=-44.332,89.625,4.399,-179.7823,0.1089,0.0000
C00591=-41.782,90.851,4.400,-179.9656,0.0172,0.0000
C00592=-39.424,91.901,4.400,-179.9943,0.0000,0.0000
C00593=-37.107,92.860,4.400,-179.9943,0.0000,0.0000
C00594=-34.697,93.786,4.400,-179.9656,0.0115,0.0000
C00595=-32.027,94.722,4.399,-179.7708,0.0745,0.0000
C00596=-29.164,95.617,4.399,-179.1806,0.2407,0.0000
C00597=-26.460,96.362,4.399,-178.2693,0.4471,0.0000
C00598=-24.268,96.890,4.398,-177.1167,0.6425,0.0000
C00599=-22.514,97.259,4.396,-175.7731,0.8388,0.0000
C00600=-20.779,97.591,4.393,-174.4382,1.0363,0.0000
C00601=-18.630,97.979,4.390,-173.2915,1.1769,0.0000
C00602=-15.506,98.490,4.388,-172.4997,1.1444,0.0000
C00603=-10.941,99.090,4.387,-172.1592,0.8618,0.0000
C00604=-5.764,99.524,4.387,-172.1138,0.4628,0.0000
C00605=0.000,99.691,4.387,-172.1025,0.0000,0.0000
C00606=0.000,99.321,6.555,-168.5271,0.0000,0.0000
C00607=5.730,99.155,6.555,-168.5440,-0.6723,0.0000
C00608=10.884,98.723,6.555,-168.6125,-1.2508,0.0000
C00609=15.437,98.140,6.558,-169.0891,-1.6049,0.0000
C00610=18.547,97.668,6.566,-170.2258,-1.5293,0.0000
C00611=20.687,97.336,6.576,-171.8926,-1.2386,0.0000
C00612=22.417,97.071,6.585,-173.8623,-0.9682,0.0000
C00613=24.167,96.770,6.592,-175.8307,-0.7870,0.0000
C00614=26.351,96.303,6.595,-177.5124,-0.5850,0.0000
C00615=29.062,95.605,6.597,-178.8311,-0.3266,0.0000
C00616=31.947,94.737,6.598,-179.6791,-0.1031,0.0000
C00617=34.646,93.803,6.599,-179.9484,-0.0172,0.0000
C00618=37.090,92.867,6.600,-179.9943,-0.0000,0.0000
C00619=39.440,91.893,6.600,-179.9943,-0.0000,0.0000
C00620=41.830,90.827,6.599,-179.9484,-0.0229,0.0000
C00621=44.399,89.579,6.598,-179.7021,-0.1547,0.0000
C00622=47.053,88.152,6.597,-178.9457,-0.5960,0.0000
C00623=49.464,86.729,6.595,-177.8216,-1.3476,0.0000
C00624=51.338,85.515,6.592,-176.4941,-2.3943,0.0000
C00625=52.788,84.491,6.585,-174.9698,-3.6664,0.0000
C00626=54.199,83.455,6.576,-173.3785,-4.8853,0.0000
C00627=55.947,82.176,6.566,-171.9913,-5.8770,0.0000
C00628=58.480,80.311,6.558,-171.1284,-6.6482,0.0000
C00629=62.112,77.504,6.555,-171.0304,-7.2336,0.0000
C00630=66.061,74.165,6.555,-171.3778,-7.6884,0.0000
C00631=70.230,70.230,6.555,-171.8355,-8.1645,0.0000
C00632=74.165,66.061,6.555,-172.3116,-8.6222,0.0000
C00633=77.504,62.112,6.555,-172.7664,-8.9696,0.0000
C00634=80.311,58.480,6.558,-173.3518,-8.8716,0.0000
C00635=82.176,55.947,6.566,-174.1230,-8.0087,0.0000
C00636=83.455,54.199,6.576,-175.1147,-6.6215,0.0000
C00637=84.491,52.788,6.585,-176.3336,-5.0302,0.0000
C00638=85.515,51.338,6.592,-177.6057,-3.5059,0.0000
C00639=86.729,49.464,6.595,-178.6524,-2.1784,0.0000
C00640=88.152,47.053,6.597,-179.4040,-1.0543,0.0000
C00641=89.579,44.399,6.598,-179.8453,-0.2979,0.0000
C00642=90.827,41.830,6.599,-179.9771,-0.0516,0.0000
C00643=91.893,39.440,6.600,-180.0000,-0.0057,0.0000
C00644=92.867,37.090,6.600,-180.0000,-0.0057,0.0000
C00645=93.803,34.646,6.599,-179.9828,-0.0516,0.0000
C00646=94.737,31.947,6.598,-179.8969,-0.3209,0.0000
C00647=95.605,29.062,6.597,-179.6734,-1.1689,0.0000
C00648=96.303,26.351,6.595,-179.4150,-2.4876,0.0000
C00649=96.770,24.167,6.592,-179.2130,-4.1693,0.0000
C00650=97.071,22.417,6.585,-179.0318,-6.1377,0.0000
C00651=97.336,20.687,6.576,-178.7614,-8.1074,0.0000
C00652=97.668,18.547,6.566,-178.4707,-9.7742,0.0000
C00653=98.140,15.437,6.558,-178.3951,-10.9109,0.0000
C00654=98.723,10.884,6.555,-178.7492,-11.3875,0.0000
C00655=99.155,5.730,6.555,-179.3277,-11.4560,0.0000
C00656=99.321,0.000,6.555,180.0000,-11.4729,0.0000
C00657=99.155,-5.730,6.555,179.3277,-11.4560,0.0000
C00658=98.723,-10.884,6.555,178.7492,-11.3875,0.0000
C00659=98.140,-15.437,6.558,178.3951,-10.9109,0.0000
C00660=97.668,-18.547,6.566,178.4707,-9.7742,0.0000
C00661=97.336,-20.687,6.576,178.7614,-8.1074,0.0000
C00662=97.071,-22.417,6.585,179.0318,-6.1377,0.0000
C00663=96.770,-24.167,6.592,179.2130,-4.1693,0.0000
C00664=96.303,-26.351,6.595,179.4150,-2.4876,0.0000
C00665=95.605,-29.062,6.597,179.6734,-1.1689,0.0000
C00666=94.737,-31.947,6.598,179.8969,-0.3209,0.0000
C00667=93.803,-34.646,6.599,179.9828,-0.0516,0.0000
C00668=92.867,-37.090,6.600,180.0000,-0.0057,0.0000
C00669=91.893,-39.440,6.600,180.0000,-0.0057,0.0000
C00670=90.827,-41.830,6.599,179.9771,-0.0516,0.0000
C00671=89.579,-44.399,6.598,179.8453,-0.2979,0.0000
C00672=88.152,-47.053,6.597,179.4040,-1.0543,0.0000
C00673=86.729,-49.464,6.595,178.6524,-2.1784,0.0000
C00674=85.515,-51.338,6.592,177.6057,-3.5059,0.0000
C00675=84.491,-52.788,6.585,176.3336,-5.0302,0.0000
C00676=83.455,-54.199,6.576,175.1147,-6.6215,0.0000
C00677=82.176,-55.947,6.566,174.1230,-8.0087,0.0000
C00678=80.311,-58.480,6.558,173.3518,-8.8716,0.0000
C00679=77.504,-62.112,6.555,172.7664,-8.9696,0.0000
C00680=74.165,-66.061,6.555,172.3116,-8.6222,0.0000
C00681=70.230,-70.230,6.555,171.8355,-8.1645,0.0000
C00682=66.061,-74.165,6.555,171.3778,-7.6884,0.0000
C00683=62.112,-77.504,6.555,171.0304,-7.2336,0.0000
C00684=58.480,-80.311,6.558,171.1284,-6.6482,0.0000
C00685=55.947,-82.176,6.566,171.9913,-5.8770,0.0000
C00686=54.199,-83.455,6.576,173.3785,-4.8853,0.0000
C00687=52.788,-84.491,6.585,174.9698,-3.6664,0.0000
C00688=51.338,-85.515,6.592,176.4941,-2.3943,0.0000
C00689=49.464,-86.729,6.595,177.8216,-1.3476,0.0000
C00690=47.053,-88.152,6.597,178.9457,-0.5960,0.0000
C00691=44.399,-89.579,6.598,179.7021,-0.1547,0.0000
C00692=41.830,-90.827,6.599,179.9484,-0.0229,0.0000
C00693=39.440,-91.893,6.600,179.9943,-0.0000,0.0000
C00694=37.090,-92.867,6.600,179.9943,-0.0000,0.0000
C00695=34.646,-93.803,6.599,179.9484,-0.0172,0.0000
C00696=31.947,-94.737,6.598,179.6791,-0.1031,0.0000
C00697=29.062,-95.605,6.597,178.8311,-0.3266,0.0000
C00698=26.351,-96.303,6.595,177.5124,-0.5850,0.0000
C00699=24.167,-96.770,6.592,175.8307,-0.7870,0.0000
C00700=22.417,-97.071,6.585,173.8623,-0.9682,0.0000
C00701=20.687,-97.336,6.576,171.8926,-1.2386,0.0000
C00702=18.547,-97.668,6.566,170.2258,-1.5293,0.0000
C00703=15.437,-98.140,6.558,169.0891,-1.6049,0.0000
C00704=10.884,-98.723,6.555,168.6125,-1.2508,0.0000
C00705=5.730,-99.155,6.555,168.5440,-0.6723,0.0000
C00706=0.000,-99.321,6.555,168.5271,0.0000,0.0000
C00707=0.000,-99.321,6.555,168.5271,0.0000,0.0000
C00708=-5.730,-99.155,6.555,168.5440,0.6723,0.0000
C00709=-10.884,-98.723,6.555,168.6125,1.2508,0.0000
C00710=-15.437,-98.140,6.558,169.0891,1.6049,0.0000
C00711=-18.547,-97.668,6.566,170.2258,1.5293,0.0000
C00712=-20.687,-97.336,6.576,171.8926,1.2386,0.0000
C00713=-22.417,-97.071,6.585,173.8623,0.9682,0.0000
C00714=-24.167,-96.770,6.592,175.8307,0.7870,0.0000
C00715=-26.351,-96.303,6.595,177.5124,0.5850,0.0000
C00716=-29.062,-95.605,6.597,178.8311,0.3266,0.0000
C00717=-31.947,-94.737,6.598,179.6791,0.1031,0.0000
C00718=-34.646,-93.803,6.599,179.9484,0.0172,0.0000
C00719=-37.090,-92.867,6.600,179.9943,0.0000,0.0000
C00720=-39.440,-91.893,6.600,179.9943,0.0000,0.0000
C00721=-41.830,-90.827,6.599,179.9484,0.0229,0.0000
C00722=-44.399,-89.579,6.598,179.7021,0.1547,0.0000
C00723=-47.053,-88.152,6.597,178.9457,0.5960,0.0000
C00724=-49.464,-86.729,6.595,177.8216,1.3476,0.0000
C00725=-51.338,-85.515,6.592,176.4941,2.3943,0.0000
C00726=-52.788,-84.491,6.585,174.9698,3.6664,0.0000
C00727=-54.199,-83.455,6.576,173.3785,4.8853,0.0000
C00728=-55.947,-82.176,6.566,171.9913,5.8770,0.0000
C00729=-58.480,-80.311,6.558,171.1284,6.6482,0.0000
C00730=-62.112,-77.504,6.555,171.0304,7.2336,0.0000
C00731=-66.061,-74.165,6.555,171.3778,7.6884,0.0000
C00732=-70.230,-70.230,6.555,171.8355,8.1645,0.0000
C00733=-74.165,-66.061,6.555,172.3116,8.6222,0.0000
C00734=-77.504,-62.112,6.555,172.7664,8.9696,0.0000
C00735=-80.311,-58.480,6.558,173.3518,8.8716,0.0000
C00736=-82.176,-55.947,6.566,174.1230,8.0087,0.0000
C00737=-83.455,-54.199,6.576,175.1147,6.6215,0.0000
C00738=-84.491,-52.788,6.585,176.3336,5.0302,0.0000
C00739=-85.515,-51.338,6.592,177.6057,3.5059,0.0000
C00740=-86.729,-49.464,6.595,178.6524,2.1784,0.0000
C00741=-88.152,-47.053,6.597,179.4040,1.0543,0.0000
C00742=-89.579,-44.399,6.598,179.8453,0.2979,0.0000
C00743=-90.827,-41.830,6.599,179.9771,0.0516,0.0000
C00744=-91.893,-39.440,6.600,180.0000,0.0057,0.0000
C00745=-92.867,-37.090,6.600,180.0000,0.0057,0.0000
C00746=-93.803,-34.646,6.599,179.9828,0.0516,0.0000
C00747=-94.737,-31.947,6.598,179.8969,0.3209,0.0000
C00748=-95.605,-29.062,6.597,179.6734,1.1689,0.0000
C00749=-96.303,-26.351,6.595,179.4150,2.4876,0.0000
C00750=-96.770,-24.167,6.592,179.2130,4.1693,0.0000
C00751=-97.071,-22.417,6.585,179.0318,6.1377,0.0000
C00752=-97.336,-20.687,6.576,178.7614,8.1074,0.0000
C00753=-97.668,-18.547,6.566,178.4707,9.7742,0.0000
C00754=-98.140,-15.437,6.558,178.3951,10.9109,0.0000
C00755=-98.723,-10.884,6.555,178.7492,11.3875,0.0000
C00756=-99.155,-5.730,6.555,179.3277,11.4560,0.0000
C00757=-99.321,0.000,6.555,-180.0000,11.4729,0.0000
C00758=-99.155,5.730,6.555,-179.3277,11.4560,0.0000
C00759=-98.723,10.884,6.555,-178.7492,11.3875,0.0000
C00760=-98.140,15.437,6.558,-178.3951,10.9109,0.0000
C00761=-97.668,18.547,6.566,-178.4707,9.7742,0.0000
C00762=-97.336,20.687,6.576,-178.7614,8.1074,0.0000
C00763=-97.071,22.417,6.585,-179.0318,6.1377,0.0000
C00764=-96.770,24.167,6.592,-179.2130,4.1693,0.0000
C00765=-96.303,26.351,6.595,-179.4150,2.4876,0.0000
C00766=-95.605,29.062,6.597,-179.6734,1.1689,0.0000
C00767=-94.737,31.947,6.598,-179.8969,0.3209,0.0000
C00768=-93.803,34.646,6.599,-179.9828,0.0516,0.0000
C00769=-92.867,37.090,6.600,-180.0000,0.0057,0.0000
C00770=-91.893,39.440,6.600,-180.0000,0.0057,0.0000
C00771=-90.827,41.830,6.599,-179.9771,0.0516,0.0000
C00772=-89.579,44.399,6.598,-179.8453,0.2979,0.0000
C00773=-88.152,47.053,6.597,-179.4040,1.0543,0.0000
C00774=-86.729,49.464,6.595,-178.6524,2.1784,0.0000
C00775=-85.515,51.338,6.592,-177.6057,3.5059,0.0000
C00776=-84.491,52.788,6.585,-176.3336,5.0302,0.0000
C00777=-83.455,54.199,6.576,-175.1147,6.6215,0.0000
C00778=-82.176,55.947,6.566,-174.1230,8.0087,0.0000
C00779=-80.311,58.480,6.558,-173.3518,8.8716,0.0000
C00780=-77.504,62.112,6.555,-172.7664,8.9696,0.0000
C00781=-74.165,66.061,6.555,-172.3116,8.6222,0.0000
C00782=-70.230,70.230,6.555,-171.8355,8.1645,0.0000
C00783=-66.061,74.165,6.555,-171.3778,7.6884,0.0000
C00784=-62.112,77.504,6.555,-171.0304,7.2336,0.0000
C00785=-58.480,80.311,6.558,-171.1284,6.6482,0.0000
C00786=-55.947,82.176,6.566,-171.9913,5.8770,0.0000
C00787=-54.199,83.455,6.576,-173.3785,4.8853,0.0000
C00788=-52.788,84.491,6.585,-174.9698,3.6664,0.0000
C00789=-51.338,85.515,6.592,-176.4941,2.3943,0.0000
C00790=-49.464,86.729,6.595,-177.8216,1.3476,0.0000
C00791=-47.053,88.152,6.597,-178.9457,0.5960,0.0000
C00792=-44.399,89.579,6.598,-179.7021,0.1547,0.0000
C00793=-41.830,90.827,6.599,-179.9484,0.0229,0.0000
C00794=-39.440,91.893,6.600,-179.9943,0.0000,0.0000
C00795=-37.090,92.867,6.600,-179.9943,0.0000,0.0000
C00796=-34.646,93.803,6.599,-179.9484,0.0172,0.0000
C00797=-31.947,94.737,6.598,-179.6791,0.1031,0.0000
C00798=-29.062,95.605,6.597,-178.8311,0.3266,0.0000
C00799=-26.351,96.303,6.595,-177.5124,0.5850,0.0000
C00800=-24.167,96.770,6.592,-175.8307,0.7870,0.0000
C00801=-22.417,97.071,6.585,-173.8623,0.9682,0.0000
C00802=-20.687,97.336,6.576,-171.8926,1.2386,0.0000
C00803=-18.547,97.668,6.566,-170.2258,1.5293,0.0000
C00804=-15.437,98.140,6.558,-169.0891,1.6049,0.0000
C00805=-10.884,98.723,6.555,-168.6125,1.2508,0.0000
C00806=-5.730,99.155,6.555,-168.5440,0.6723,0.0000
C00807=0.000,99.321,6.555,-168.5271,0.0000,0.0000
C00808=0.000,98.820,8.697,-165.2384,0.0000,0.0000
C00809=5.684,98.656,8.697,-165.2550,-0.8768,0.0000
C00810=10.807,98.229,8.698,-165.3451,-1.6051,0.0000
C00811=15.344,97.668,8.705,-165.9346,-1.9495,0.0000
C00812=18.436,97.247,8.723,-167.3804,-1.6441,0.0000
C00813=20.563,96.991,8.745,-169.5521,-1.1187,0.0000
C00814=22.286,96.814,8.767,-172.1365,-0.8040,0.0000
C00815=24.029,96.606,8.782,-174.6920,-0.7538,0.0000
C00816=26.202,96.222,8.789,-176.8469,-0.6485,0.0000
C00817=28.922,95.588,8.792,-178.5388,-0.3783,0.0000
C00818=31.837,94.757,8.795,-179.6161,-0.1203,0.0000
C00819=34.577,93.826,8.798,-179.9370,-0.0229,0.0000
C00820=37.066,92.876,8.800,-179.9943,-0.0057,0.0000
C00821=39.463,91.883,8.800,-179.9943,-0.0057,0.0000
C00822=41.895,90.794,8.798,-179.9370,-0.0286,0.0000
C00823=44.491,89.515,8.795,-179.6448,-0.1891,0.0000
C00824=47.140,88.042,8.792,-178.6992,-0.7622,0.0000
C00825=49.511,86.567,8.789,-177.3105,-1.7727,0.0000
C00826=51.320,85.302,8.782,-175.7091,-3.2251,0.0000
C00827=52.699,84.217,8.767,-173.8631,-5.0139,0.0000
C00828=54.043,83.124,8.745,-171.7932,-6.6483,0.0000
C00829=55.728,81.800,8.723,-169.8751,-7.8561,0.0000
C00830=58.212,79.911,8.705,-168.6219,-8.7026,0.0000
C00831=61.817,77.101,8.698,-168.4294,-9.3768,0.0000
C00832=65.741,73.780,8.697,-168.8611,-9.9421,0.0000
C00833=69.877,69.877,8.697,-169.4440,-10.5560,0.0000
C00834=73.780,65.741,8.697,-170.0579,-11.1389,0.0000
C00835=77.101,61.817,8.698,-170.6232,-11.5706,0.0000
C00836=79.911,58.212,8.705,-171.2974,-11.3781,0.0000
C00837=81.800,55.728,8.723,-172.1439,-10.1249,0.0000
C00838=83.124,54.043,8.745,-173.3517,-8.2068,0.0000
C00839=84.217,52.699,8.767,-174.9861,-6.1369,0.0000
C00840=85.302,51.320,8.782,-176.7749,-4.2909,0.0000
C00841=86.567,49.511,8.789,-178.2273,-2.6895,0.0000
C00842=88.042,47.140,8.792,-179.2378,-1.3008,0.0000
C00843=89.515,44.491,8.795,-179.8109,-0.3552,0.0000
C00844=90.794,41.895,8.798,-179.9714,-0.0630,0.0000
C00845=91.883,39.463,8.800,-179.9943,-0.0057,0.0000
C00846=92.876,37.066,8.800,-179.9943,-0.0057,0.0000
C00847=93.826,34.577,8.798,-179.9771,-0.0630,0.0000
C00848=94.757,31.837,8.795,-179.8797,-0.3839,0.0000
C00849=95.588,28.922,8.792,-179.6217,-1.4612,0.0000
C00850=96.222,26.202,8.789,-179.3515,-3.1531,0.0000
C00851=96.606,24.029,8.782,-179.2462,-5.3080,0.0000
C00852=96.814,22.286,8.767,-179.1960,-7.8635,0.0000
C00853=96.991,20.563,8.745,-178.8813,-10.4479,0.0000
C00854=97.247,18.436,8.723,-178.3559,-12.6196,0.0000
C00855=97.668,15.344,8.705,-178.0505,-14.0654,0.0000
C00856=98.229,10.807,8.698,-178.3949,-14.6549,0.0000
C00857=98.656,5.684,8.697,-179.1232,-14.7450,0.0000
C00858=98.820,0.000,8.697,180.0000,-14.7616,0.0000
C00859=98.656,-5.684,8.697,179.1232,-14.7450,0.0000
C00860=98.229,-10.807,8.698,178.3949,-14.6549,0.0000
C00861=97.668,-15.344,8.705,178.0505,-14.0654,0.0000
C00862=97.247,-18.436,8.723,178.3559,-12.6196,0.0000
C00863=96.991,-20.563,8.745,178.8813,-10.4479,0.0000
C00864=96.814,-22.286,8.767,179.1960,-7.8635,0.0000
C00865=96.606,-24.029,8.782,179.2462,-5.3080,0.0000
C00866=96.222,-26.202,8.789,179.3515,-3.1531,0.0000
C00867=95.588,-28.922,8.792,179.6217,-1.4612,0.0000
C00868=94.757,-31.837,8.795,179.8797,-0.3839,0.0000
C00869=93.826,-34.577,8.798,179.9771,-0.0630,0.0000
C00870=92.876,-37.066,8.800,179.9943,-0.0057,0.0000
C00871=91.883,-39.463,8.800,179.9943,-0.0057,0.0000
C00872=90.794,-41.895,8.798,179.9714,-0.0630,0.0000
C00873=89.515,-44.491,8.795,179.8109,-0.3552,0.0000
C00874=88.042,-47.140,8.792,179.2378,-1.3008,0.0000
C00875=86.567,-49.511,8.789,178.2273,-2.6895,0.0000
C00876=85.302,-51.320,8.782,176.7749,-4.2909,0.0000
C00877=84.217,-52.699,8.767,174.9861,-6.1369,0.0000
C00878=83.124,-54.043,8.745,173.3517,-8.2068,0.0000
C00879=81.800,-55.728,8.723,172.1439,-10.1249,0.0000
C00880=79.911,-58.212,8.705,171.2974,-11.3781,0.0000
C00881=77.101,-61.817,8.698,170.6232,-11.5706,0.0000
C00882=73.780,-65.741,8.697,170.0579,-11.1389,0.0000
C00883=69.877,-69.877,8.697,169.4440,-10.5560,0.0000
C00884=65.741,-73.780,8.697,168.8611,-9.9421,0.0000
C00885=61.817,-77.101,8.698,168.4294,-9.3768,0.0000
C00886=58.212,-79.911,8.705,168.6219,-8.7026,0.0000
C00887=55.728,-81.800,8.723,169.8751,-7.8561,0.0000
C00888=54.043,-83.124,8.745,171.7932,-6.6483,0.0000
C00889=52.699,-84.217,8.767,173.8631,-5.0139,0.0000
C00890=51.320,-85.302,8.782,175.7091,-3.2251,0.0000
C00891=49.511,-86.567,8.789,177.3105,-1.7727,0.0000
C00892=47.140,-88.042,8.792,178.6992,-0.7622,0.0000
C00893=44.491,-89.515,8.795,179.6448,-0.1891,0.0000
C00894=41.895,-90.794,8.798,179.9370,-0.0286,0.0000
C00895=39.463,-91.883,8.800,179.9943,-0.0057,0.0000
C00896=37.066,-92.876,8.800,179.9943,-0.0057,0.0000
C00897=34.577,-93.826,8.798,179.9370,-0.0229,0.0000
C00898=31.837,-94.757,8.795,179.6161,-0.1203,0.0000
C00899=28.922,-95.588,8.792,178.5388,-0.3783,0.0000
C00900=26.202,-96.222,8.789,176.8469,-0.6485,0.0000
C00901=24.029,-96.606,8.782,174.6920,-0.7538,0.0000
C00902=22.286,-96.814,8.767,172.1365,-0.8040,0.0000
C00903=20.563,-96.991,8.745,169.5521,-1.1187,0.0000
C00904=18.436,-97.247,8.723,167.3804,-1.6441,0.0000
C00905=15.344,-97.668,8.705,165.9346,-1.9495,0.0000
C00906=10.807,-98.229,8.698,165.3451,-1.6051,0.0000
C00907=5.684,-98.656,8.697,165.2550,-0.8768,0.0000
C00908=0.000,-98.820,8.697,165.2384,0.0000,0.0000
C00909=0.000,-98.820,8.697,165.2384,0.0000,0.0000
C00910=-5.684,-98.656,8.697,165.2550,0.8768,0.0000
C00911=-10.807,-98.229,8.698,165.3451,1.6051,0.0000
C00912=-15.344,-97.668,8.705,165.9346,1.9495,0.0000
C00913=-18.436,-97.247,8.723,167.3804,1.6441,0.0000
C00914=-20.563,-96.991,8.745,169.5521,1.1187,0.0000
C00915=-22.286,-96.814,8.767,172.1365,0.8040,0.0000
C00916=-24.029,-96.606,8.782,174.6920,0.7538,0.0000
C00917=-26.202,-96.222,8.789,176.8469,0.6485,0.0000
C00918=-28.922,-95.588,8.792,178.5388,0.3783,0.0000
C00919=-31.837,-94.757,8.795,179.6161,0.1203,0.0000
C00920=-34.577,-93.826,8.798,179.9370,0.0229,0.0000
C00921=-37.066,-92.876,8.800,179.9943,0.0057,0.0000
C00922=-39.463,-91.883,8.800,179.9943,0.0057,0.0000
C00923=-41.895,-90.794,8.798,179.9370,0.0286,0.0000
C00924=-44.491,-89.515,8.795,179.6448,0.1891,0.0000
C00925=-47.140,-88.042,8.792,178.6992,0.7622,0.0000
C00926=-49.511,-86.567,8.789,177.3105,1.7727,0.0000
C00927=-51.320,-85.302,8.782,175.7091,3.2251,0.0000
C00928=-52.699,-84.217,8.767,173.8631,5.0139,0.0000
C00929=-54.043,-83.124,8.745,171.7932,6.6483,0.0000
C00930=-55.728,-81.800,8.723,169.8751,7.8561,0.0000
C00931=-58.212,-79.911,8.705,168.6219,8.7026,0.0000
C00932=-61.817,-77.101,8.698,168.4294,9.3768,0.0000
C00933=-65.741,-73.780,8.697,168.8611,9.9421,0.0000
C00934=-69.877,-69.877,8.697,169.4440,10.5560,0.0000
C00935=-73.780,-65.741,8.697,170.0579,11.1389,0.0000
C00936=-77.101,-61.817,8.698,170.6232,11.5706,0.0000
C00937=-79.911,-58.212,8.705,171.2974,11.3781,0.0000
C00938=-81.800,-55.728,8.723,172.1439,10.1249,0.0000
C00939=-83.124,-54.043,8.745,173.3517,8.2068,0.0000
C00940=-84.217,-52.699,8.767,174.9861,6.1369,0.0000
C00941=-85.302,-51.320,8.782,176.7749,4.2909,0.0000
C00942=-86.567,-49.511,8.789,178.2273,2.6895,0.0000
C00943=-88.042,-47.140,8.792,179.2378,1.3008,0.0000
C00944=-89.515,-44.491,8.795,179.8109,0.3552,0.0000
C00945=-90.794,-41.895,8.798,179.9714,0.0630,0.0000
C00946=-91.883,-39.463,8.800,179.9943,0.0057,0.0000
C00947=-92.876,-37.066,8.800,179.9943,0.0057,0.0000
C00948=-93.826,-34.577,8.798,179.9771,0.0630,0.0000
C00949=-94.757,-31.837,8.795,179.8797,0.3839,0.0000
C00950=-95.588,-28.922,8.792,179.6217,1.4612,0.0000
C00951=-96.222,-26.202,8.789,179.3515,3.1531,0.0000
C00952=-96.606,-24.029,8.782,179.2462,5.3080,0.0000
C00953=-96.814,-22.286,8.767,179.1960,7.8635,0.0000
C00954=-96.991,-20.563,8.745,178.8813,10.4479,0.0000
C00955=-97.247,-18.436,8.723,178.3559,12.6196,0.0000
C00956=-97.668,-15.344,8.705,178.0505,14.0654,0.0000
C00957=-98.229,-10.807,8.698,178.3949,14.6549,0.0000
C00958=-98.656,-5.684,8.697,179.1232,14.7450,0.0000
C00959=-98.820,0.000,8.697,-180.0000,14.7616,0.0000
C00960=-98.656,5.684,8.697,-179.1232,14.7450,0.0000
C00961=-98.229,10.807,8.698,-178.3949,14.6549,0.0000
C00962=-97.668,15.344,8.705,-178.0505,14.0654,0.0000
C00963=-97.247,18.436,8.723,-178.3559,12.6196,0.0000
C00964=-96.991,20.563,8.745,-178.8813,10.4479,0.0000
C00965=-96.814,22.286,8.767,-179.1960,7.8635,0.0000
C00966=-96.606,24.029,8.782,-179.2462,5.3080,0.0000
C00967=-96.222,26.202,8.789,-179.3515,3.1531,0.0000
C00968=-95.588,28.922,8.792,-179.6217,1.4612,0.0000
C00969=-94.757,31.837,8.795,-179.8797,0.3839,0.0000
C00970=-93.826,34.577,8.798,-179.9771,0.0630,0.0000
C00971=-92.876,37.066,8.800,-179.9943,0.0057,0.0000
C00972=-91.883,39.463,8.800,-179.9943,0.0057,0.0000
C00973=-90.794,41.895,8.798,-179.9714,0.0630,0.0000
C00974=-89.515,44.491,8.795,-179.8109,0.3552,0.0000
C00975=-88.042,47.140,8.792,-179.2378,1.3008,0.0000
C00976=-86.567,49.511,8.789,-178.2273,2.6895,0.0000
C00977=-85.302,51.320,8.782,-176.7749,4.2909,0.0000
C00978=-84.217,52.699,8.767,-174.9861,6.1369,0.0000
C00979=-83.124,54.043,8.745,-173.3517,8.2068,0.0000
C00980=-81.800,55.728,8.723,-172.1439,10.1249,0.0000
C00981=-79.911,58.212,8.705,-171.2974,11.3781,0.0000
C00982=-77.101,61.817,8.698,-170.6232,11.5706,0.0000
C00983=-73.780,65.741,8.697,-170.0579,11.1389,0.0000
C00984=-69.877,69.877,8.697,-169.4440,10.5560,0.0000
C00985=-65.741,73.780,8.697,-168.8611,9.9421,0.0000
C00986=-61.817,77.101,8.698,-168.4294,9.3768,0.0000
C00987=-58.212,79.911,8.705,-168.6219,8.7026,0.0000
C00988=-55.728,81.800,8.723,-169.8751,7.8561,0.0000
C00989=-54.043,83.124,8.745,-171.7932,6.6483,0.0000
C00990=-52.699,84.217,8.767,-173.8631,5.0139,0.0000
C00991=-51.320,85.302,8.782,-175.7091,3.2251,0.0000
C00992=-49.511,86.567,8.789,-177.3105,1.7727,0.0000
C00993=-47.140,88.042,8.792,-178.6992,0.7622,0.0000
C00994=-44.491,89.515,8.795,-179.6448,0.1891,0.0000
C00995=-41.895,90.794,8.798,-179.9370,0.0286,0.0000
C00996=-39.463,91.883,8.800,-179.9943,0.0057,0.0000
C00997=-37.066,92.876,8.800,-179.9943,0.0057,0.0000
C00998=-34.577,93.826,8.798,-179.9370,0.0229,0.0000
C00999=-31.837,94.757,8.795,-179.6161,0.1203,0.0000
C01000=-28.922,95.588,8.792,-178.5388,0.3783,0.0000
C01001=-26.202,96.222,8.789,-176.8469,0.6485,0.0000
C01002=-24.029,96.606,8.782,-174.6920,0.7538,0.0000
C01003=-22.286,96.814,8.767,-172.1365,0.8040,0.0000
C01004=-20.563,96.991,8.745,-169.5521,1.1187,0.0000
C01005=-18.436,97.247,8.723,-167.3804,1.6441,0.0000
C01006=-15.344,97.668,8.705,-165.9346,1.9495,0.0000
C01007=-10.807,98.229,8.698,-165.3451,1.6051,0.0000
C01008=-5.684,98.656,8.697,-165.2550,0.8768,0.0000
C01009=0.000,98.820,8.697,-165.2384,0.0000,0.0000
C01010=0.000,98.204,10.809,-162.2409,0.0000,0.0000
C01011=5.628,98.041,10.809,-162.2573,-1.0588,0.0000
C01012=10.712,97.620,10.809,-162.3591,-1.9122,0.0000
C01013=15.229,97.084,10.823,-163.0465,-2.1688,0.0000
C01014=18.298,96.727,10.856,-164.7821,-1.4728,0.0000
C01015=20.409,96.562,10.898,-167.4898,-0.6162,0.0000
C01016=22.123,96.495,10.937,-170.6940,-0.2903,0.0000
C01017=23.856,96.400,10.965,-173.7478,-0.5188,0.0000
C01018=26.016,96.121,10.978,-176.3075,-0.6201,0.0000
C01019=28.748,95.567,10.985,-178.3209,-0.3955,0.0000
C01020=31.699,94.782,10.991,-179.5817,-0.1261,0.0000
C01021=34.490,93.854,10.996,-179.9255,-0.0286,0.0000
C01022=37.037,92.887,11.000,-179.9943,-0.0057,0.0000
C01023=39.492,91.870,11.000,-179.9943,-0.0057,0.0000
C01024=41.977,90.753,10.996,-179.9312,-0.0344,0.0000
C01025=44.606,89.436,10.991,-179.6161,-0.2063,0.0000
C01026=47.248,87.904,10.985,-178.5328,-0.9114,0.0000
C01027=49.571,86.364,10.978,-176.9483,-2.1750,0.0000
C01028=51.296,85.034,10.965,-175.2039,-4.0627,0.0000
C01029=52.589,83.875,10.937,-173.1868,-6.4065,0.0000
C01030=53.849,82.711,10.898,-170.6634,-8.4889,0.0000
C01031=55.458,81.334,10.856,-168.1098,-9.8798,0.0000
C01032=57.880,79.417,10.823,-166.3749,-10.6873,0.0000
C01033=61.453,76.603,10.809,-166.0445,-11.3793,0.0000
C01034=65.346,73.305,10.809,-166.5414,-12.0335,0.0000
C01035=69.440,69.440,10.809,-167.2376,-12.7624,0.0000
C01036=73.305,65.346,10.809,-167.9665,-13.4586,0.0000
C01037=76.603,61.453,10.809,-168.6207,-13.9555,0.0000
C01038=79.417,57.880,10.823,-169.3127,-13.6251,0.0000
C01039=81.334,55.458,10.856,-170.1202,-11.8902,0.0000
C01040=82.711,53.849,10.898,-171.5111,-9.3366,0.0000
C01041=83.875,52.589,10.937,-173.5935,-6.8132,0.0000
C01042=85.034,51.296,10.965,-175.9373,-4.7961,0.0000
C01043=86.364,49.571,10.978,-177.8250,-3.0517,0.0000
C01044=87.904,47.248,10.985,-179.0886,-1.4672,0.0000
C01045=89.436,44.606,10.991,-179.7937,-0.3839,0.0000
C01046=90.753,41.977,10.996,-179.9656,-0.0688,0.0000
C01047=91.870,39.492,11.000,-179.9943,-0.0057,0.0000
C01048=92.887,37.037,11.000,-179.9943,-0.0057,0.0000
C01049=93.854,34.490,10.996,-179.9714,-0.0745,0.0000
C01050=94.782,31.699,10.991,-179.8739,-0.4183,0.0000
C01051=95.567,28.748,10.985,-179.6045,-1.6791,0.0000
C01052=96.121,26.016,10.978,-179.3799,-3.6925,0.0000
C01053=96.400,23.856,10.965,-179.4812,-6.2522,0.0000
C01054=96.495,22.123,10.937,-179.7097,-9.3060,0.0000
C01055=96.562,20.409,10.898,-179.3838,-12.5102,0.0000
C01056=96.727,18.298,10.856,-178.5272,-15.2179,0.0000
C01057=97.084,15.229,10.823,-177.8312,-16.9535,0.0000
C01058=97.620,10.712,10.809,-178.0878,-17.6409,0.0000
C01059=98.041,5.628,10.809,-178.9412,-17.7427,0.0000
C01060=98.204,0.000,10.809,180.0000,-17.7591,0.0000
C01061=98.041,-5.628,10.809,178.9412,-17.7427,0.0000
C01062=97.620,-10.712,10.809,178.0878,-17.6409,0.0000
C01063=97.084,-15.229,10.823,177.8312,-16.9535,0.0000
C01064=96.727,-18.298,10.856,178.5272,-15.2179,0.0000
C01065=96.562,-20.409,10.898,179.3838,-12.5102,0.0000
C01066=96.495,-22.123,10.937,179.7097,-9.3060,0.0000
C01067=96.400,-23.856,10.965,179.4812,-6.2522,0.0000
C01068=96.121,-26.016,10.978,179.3799,-3.6925,0.0000
C01069=95.567,-28.748,10.985,179.6045,-1.6791,0.0000
C01070=94.782,-31.699,10.991,179.8739,-0.4183,0.0000
C01071=93.854,-34.490,10.996,179.9714,-0.0745,0.0000
C01072=92.887,-37.037,11.000,179.9943,-0.0057,0.0000
C01073=91.870,-39.492,11.000,179.9943,-0.0057,0.0000
C01074=90.753,-41.977,10.996,179.9656,-0.0688,0.0000
C01075=89.436,-44.606,10.991,179.7937,-0.3839,0.0000
C01076=87.904,-47.248,10.985,179.0886,-1.4672,0.0000
C01077=86.364,-49.571,10.978,177.8250,-3.0517,0.0000
C01078=85.034,-51.296,10.965,175.9373,-4.7961,0.0000
C01079=83.875,-52.589,10.937,173.5935,-6.8132,0.0000
C01080=82.711,-53.849,10.898,171.5111,-9.3366,0.0000
C01081=81.334,-55.458,10.856,170.1202,-11.8902,0.0000
C01082=79.417,-57.880,10.823,169.3127,-13.6251,0.0000
C01083=76.603,-61.453,10.809,168.6207,-13.9555,0.0000
C01084=73.305,-65.346,10.809,167.9665,-13.4586,0.0000
C01085=69.440,-69.440,10.809,167.2376,-12.7624,0.0000
C01086=65.346,-73.305,10.809,166.5414,-12.0335,0.0000
C01087=61.453,-76.603,10.809,166.0445,-11.3793,0.0000
C01088=57.880,-79.417,10.823,166.3749,-10.6873,0.0000
C01089=55.458,-81.334,10.856,168.1098,-9.8798,0.0000
C01090=53.849,-82.711,10.898,170.6634,-8.4889,0.0000
C01091=52.589,-83.875,10.937,173.1868,-6.4065,0.0000
C01092=51.296,-85.034,10.965,175.2039,-4.0627,0.0000
C01093=49.571,-86.364,10.978,176.9483,-2.1750,0.0000
C01094=47.248,-87.904,10.985,178.5328,-0.9114,0.0000
C01095=44.606,-89.436,10.991,179.6161,-0.2063,0.0000
C01096=41.977,-90.753,10.996,179.9312,-0.0344,0.0000
C01097=39.492,-91.870,11.000,179.9943,-0.0057,0.0000
C01098=37.037,-92.887,11.000,179.9943,-0.0057,0.0000
C01099=34.490,-93.854,10.996,179.9255,-0.0286,0.0000
C01100=31.699,-94.782,10.991,179.5817,-0.1261,0.0000
C01101=28.748,-95.567,10.985,178.3209,-0.3955,0.0000
C01102=26.016,-96.121,10.978,176.3075,-0.6201,0.0000
C01103=23.856,-96.400,10.965,173.7478,-0.5188,0.0000
C01104=22.123,-96.495,10.937,170.6940,-0.2903,0.0000
C01105=20.409,-96.562,10.898,167.4898,-0.6162,0.0000
C01106=18.298,-96.727,10.856,164.7821,-1.4728,0.0000
C01107=15.229,-97.084,10.823,163.0465,-2.1688,0.0000
C01108=10.712,-97.620,10.809,162.3591,-1.9122,0.0000
C01109=5.628,-98.041,10.809,162.2573,-1.0588,0.0000
C01110=0.000,-98.204,10.809,162.2409,0.0000,0.0000
C01111=0.000,-98.204,10.809,162.2409,0.0000,0.0000
C01112=-5.628,-98.041,10.809,162.2573,1.0588,0.0000
C01113=-10.712,-97.620,10.809,162.3591,1.9122,0.0000
C01114=-15.229,-97.084,10.823,163.0465,2.1688,0.0000
C01115=-18.298,-96.727,10.856,164.7821,1.4728,0.0000
C01116=-20.409,-96.562,10.898,167.4898,0.6162,0.0000
C01117=-22.123,-96.495,10.937,170.6940,0.2903,0.0000
C01118=-23.856,-96.400,10.965,173.7478,0.5188,0.0000
C01119=-26.016,-96.121,10.978,176.3075,0.6201,0.0000
C01120=-28.748,-95.567,10.985,178.3209,0.3955,0.0000
C01121=-31.699,-94.782,10.991,179.5817,0.1261,0.0000
C01122=-34.490,-93.854,10.996,179.9255,0.0286,0.0000
C01123=-37.037,-92.887,11.000,179.9943,0.0057,0.0000
C01124=-39.492,-91.870,11.000,179.9943,0.0057,0.0000
C01125=-41.977,-90.753,10.996,179.9312,0.0344,0.0000
C01126=-44.606,-89.436,10.991,179.6161,0.2063,0.0000
C01127=-47.248,-87.904,10.985,178.5328,0.9114,0.0000
C01128=-49.571,-86.364,10.978,176.9483,2.1750,0.0000
C01129=-51.296,-85.034,10.965,175.2039,4.0627,0.0000
C01130=-52.589,-83.875,10.937,173.1868,6.4065,0.0000
C01131=-53.849,-82.711,10.898,170.6634,8.4889,0.0000
C01132=-55.458,-81.334,10.856,168.1098,9.8798,0.0000
C01133=-57.880,-79.417,10.823,166.3749,10.6873,0.0000
C01134=-61.453,-76.603,10.809,166.0445,11.3793,0.0000
C01135=-65.346,-73.305,10.809,166.5414,12.0335,0.0000
C01136=-69.440,-69.440,10.809,167.2376,12.7624,0.0000
C01137=-73.305,-65.346,10.809,167.9665,13.4586,0.0000
C01138=-76.603,-61.453,10.809,168.6207,13.9555,0.0000
C01139=-79.417,-57.880,10.823,169.3127,13.6251,0.0000
C01140=-81.334,-55.458,10.856,170.1202,11.8902,0.0000
C01141=-82.711,-53.849,10.898,171.5111,9.3366,0.0000
C01142=-83.875,-52.589,10.937,173.5935,6.8132,0.0000
C01143=-85.034,-51.296,10.965,175.9373,4.7961,0.0000
C01144=-86.364,-49.571,10.978,177.8250,3.0517,0.0000
C01145=-87.904,-47.248,10.985,179.0886,1.4672,0.0000
C01146=-89.436,-44.606,10.991,179.7937,0.3839,0.0000
C01147=-90.753,-41.977,10.996,179.9656,0.0688,0.0000
C01148=-91.870,-39.492,11.000,179.9943,0.0057,0.0000
C01149=-92.887,-37.037,11.000,179.9943,0.0057,0.0000
C01150=-93.854,-34.490,10.996,179.9714,0.0745,0.0000
C01151=-94.782,-31.699,10.991,179.8739,0.4183,0.0000
C01152=-95.567,-28.748,10.985,179.6045,1.6791,0.0000
C01153=-96.121,-26.016,10.978,179.3799,3.6925,0.0000
C01154=-96.400,-23.856,10.965,179.4812,6.2522,0.0000
C01155=-96.495,-22.123,10.937,179.7097,9.3060,0.0000
C01156=-96.562,-20.409,10.898,179.3838,12.5102,0.0000
C01157=-96.727,-18.298,10.856,178.5272,15.2179,0.0000
C01158=-97.084,-15.229,10.823,177.8312,16.9535,0.0000
C01159=-97.620,-10.712,10.809,178.0878,17.6409,0.0000
C01160=-98.041,-5.628,10.809,178.9412,17.7427,0.0000
C01161=-98.204,0.000,10.809,-180.0000,17.7591,0.0000
C01162=-98.041,5.628,10.809,-178.9412,17.7427,0.0000
C01163=-97.620,10.712,10.809,-178.0878,17.6409,0.0000
C01164=-97.084,15.229,10.823,-177.8312,16.9535,0.0000
C01165=-96.727,18.298,10.856,-178.5272,15.2179,0.0000
C01166=-96.562,20.409,10.898,-179.3838,12.5102,0.0000
C01167=-96.495,22.123,10.937,-179.7097,9.3060,0.0000
C01168=-96.400,23.856,10.965,-179.4812,6.2522,0.0000
C01169=-96.121,26.016,10.978,-179.3799,3.6925,0.0000
C01170=-95.567,28.748,10.985,-179.6045,1.6791,0.0000
C01171=-94.782,31.699,10.991,-179.8739,0.4183,0.0000
C01172=-93.854,34.490,10.996,-179.9714,0.0745,0.0000
C01173=-92.887,37.037,11.000,-179.9943,0.0057,0.0000
C01174=-91.870,39.492,11.000,-179.9943,0.0057,0.0000
C01175=-90.753,41.977,10.996,-179.9656,0.0688,0.0000
C01176=-89.436,44.606,10.991,-179.7937,0.3839,0.0000
C01177=-87.904,47.248,10.985,-179.0886,1.4672,0.0000
C01178=-86.364,49.571,10.978,-177.8250,3.0517,0.0000
C01179=-85.034,51.296,10.965,-175.9373,4.7961,0.0000
C01180=-83.875,52.589,10.937,-173.5935,6.8132,0.0000
C01181=-82.711,53.849,10.898,-171.5111,9.3366,0.0000
C01182=-81.334,55.458,10.856,-170.1202,11.8902,0.0000
C01183=-79.417,57.880,10.823,-169.3127,13.6251,0.0000
C01184=-76.603,61.453,10.809,-168.6207,13.9555,0.0000
C01185=-73.305,65.346,10.809,-167.9665,13.4586,0.0000
C01186=-69.440,69.440,10.809,-167.2376,12.7624,0.0000
C01187=-65.346,73.305,10.809,-166.5414,12.0335,0.0000
C01188=-61.453,76.603,10.809,-166.0445,11.3793,0.0000
C01189=-57.880,79.417,10.823,-166.3749,10.6873,0.0000
C01190=-55.458,81.334,10.856,-168.1098,9.8798,0.0000
C01191=-53.849,82.711,10.898,-170.6634,8.4889,0.0000
C01192=-52.589,83.875,10.937,-173.1868,6.4065,0.0000
C01193=-51.296,85.034,10.965,-175.2039,4.0627,0.0000
C01194=-49.571,86.364,10.978,-176.9483,2.1750,0.0000
C01195=-47.248,87.904,10.985,-178.5328,0.9114,0.0000
C01196=-44.606,89.436,10.991,-179.6161,0.2063,0.0000
C01197=-41.977,90.753,10.996,-179.9312,0.0344,0.0000
C01198=-39.492,91.870,11.000,-179.9943,0.0057,0.0000
C01199=-37.037,92.887,11.000,-179.9943,0.0057,0.0000
C01200=-34.490,93.854,10.996,-179.9255,0.0286,0.0000
C01201=-31.699,94.782,10.991,-179.5817,0.1261,0.0000
C01202=-28.748,95.567,10.985,-178.3209,0.3955,0.0000
C01203=-26.016,96.121,10.978,-176.3075,0.6201,0.0000
C01204=-23.856,96.400,10.965,-173.7478,0.5188,0.0000
C01205=-22.123,96.495,10.937,-170.6940,0.2903,0.0000
C01206=-20.409,96.562,10.898,-167.4898,0.6162,0.0000
C01207=-18.298,96.727,10.856,-164.7821,1.4728,0.0000
C01208=-15.229,97.084,10.823,-163.0465,2.1688,0.0000
C01209=-10.712,97.620,10.809,-162.3591,1.9122,0.0000
C01210=-5.628,98.041,10.809,-162.2573,1.0588,0.0000
C01211=0.000,98.204,10.809,-162.2409,0.0000,0.0000
C01212=0.000,97.482,12.888,-159.5244,0.0000,0.0000
C01213=5.562,97.322,12.887,-159.5459,-1.2353,0.0000
C01214=10.602,96.908,12.888,-159.6573,-2.1819,0.0000
C01215=15.094,96.401,12.910,-160.4245,-2.2505,0.0000
C01216=18.135,96.115,12.963,-162.4730,-0.9855,0.0000
C01217=20.227,96.057,13.031,-165.7998,0.3014,0.0000
C01218=21.929,96.117,13.096,-169.6352,0.5534,0.0000
C01219=23.652,96.157,13.142,-173.0619,-0.0808,0.0000
C01220=25.795,96.000,13.164,-175.9054,-0.5055,0.0000
C01221=28.540,95.542,13.175,-178.1720,-0.3783,0.0000
C01222=31.535,94.812,13.184,-179.5703,-0.1203,0.0000
C01223=34.387,93.888,13.193,-179.9255,-0.0286,0.0000
C01224=37.002,92.901,13.199,-179.9885,-0.0057,0.0000
C01225=39.526,91.855,13.199,-179.9885,-0.0057,0.0000
C01226=42.074,90.704,13.193,-179.9255,-0.0344,0.0000
C01227=44.743,89.341,13.184,-179.6104,-0.2177,0.0000
C01228=47.377,87.740,13.175,-178.4412,-1.0260,0.0000
C01229=49.643,86.123,13.164,-176.7464,-2.5431,0.0000
C01230=51.269,84.717,13.142,-175.0258,-4.8596,0.0000
C01231=52.459,83.471,13.096,-173.0155,-7.7579,0.0000
C01232=53.620,82.225,13.031,-170.0591,-10.3532,0.0000
C01233=55.140,80.787,12.963,-166.7498,-11.9280,0.0000
C01234=57.492,78.839,12.910,-164.3984,-12.6087,0.0000
C01235=61.028,76.021,12.888,-163.8747,-13.2364,0.0000
C01236=64.884,72.750,12.887,-164.4147,-13.9556,0.0000
C01237=68.930,68.930,12.888,-165.2122,-14.7878,0.0000
C01238=72.750,64.884,12.887,-166.0444,-15.5853,0.0000
C01239=76.021,61.028,12.888,-166.7636,-16.1253,0.0000
C01240=78.839,57.492,12.910,-167.3913,-15.6016,0.0000
C01241=80.787,55.140,12.963,-168.0720,-13.2502,0.0000
C01242=82.225,53.620,13.031,-169.6468,-9.9409,0.0000
C01243=83.471,52.459,13.096,-172.2421,-6.9845,0.0000
C01244=84.717,51.269,13.142,-175.1404,-4.9742,0.0000
C01245=86.123,49.643,13.164,-177.4569,-3.2536,0.0000
C01246=87.740,47.377,13.175,-178.9740,-1.5588,0.0000
C01247=89.341,44.743,13.184,-179.7823,-0.3896,0.0000
C01248=90.704,42.074,13.193,-179.9656,-0.0745,0.0000
C01249=91.855,39.526,13.199,-179.9943,-0.0115,0.0000
C01250=92.901,37.002,13.199,-179.9943,-0.0115,0.0000
C01251=93.888,34.387,13.193,-179.9714,-0.0745,0.0000
C01252=94.812,31.535,13.184,-179.8797,-0.4297,0.0000
C01253=95.542,28.540,13.175,-179.6217,-1.8280,0.0000
C01254=96.000,25.795,13.164,-179.4945,-4.0946,0.0000
C01255=96.157,23.652,13.142,-179.9192,-6.9381,0.0000
C01256=96.117,21.929,13.096,179.4466,-10.3648,0.0000
C01257=96.057,20.227,13.031,179.6986,-14.2002,0.0000
C01258=96.115,18.135,12.963,-179.0145,-17.5270,0.0000
C01259=96.401,15.094,12.910,-177.7495,-19.5755,0.0000
C01260=96.908,10.602,12.888,-177.8181,-20.3427,0.0000
C01261=97.322,5.562,12.887,-178.7647,-20.4541,0.0000
C01262=97.482,0.000,12.888,180.0000,-20.4756,0.0000
C01263=97.322,-5.562,12.887,178.7647,-20.4541,0.0000
C01264=96.908,-10.602,12.888,177.8181,-20.3427,0.0000
C01265=96.401,-15.094,12.910,177.7495,-19.5755,0.0000
C01266=96.115,-18.135,12.963,179.0145,-17.5270,0.0000
C01267=96.057,-20.227,13.031,-179.6986,-14.2002,0.0000
C01268=96.117,-21.929,13.096,-179.4466,-10.3648,0.0000
C01269=96.157,-23.652,13.142,179.9192,-6.9381,0.0000
C01270=96.000,-25.795,13.164,179.4945,-4.0946,0.0000
C01271=95.542,-28.540,13.175,179.6217,-1.8280,0.0000
C01272=94.812,-31.535,13.184,179.8797,-0.4297,0.0000
C01273=93.888,-34.387,13.193,179.9714,-0.0745,0.0000
C01274=92.901,-37.002,13.199,179.9943,-0.0115,0.0000
C01275=91.855,-39.526,13.199,179.9943,-0.0115,0.0000
C01276=90.704,-42.074,13.193,179.9656,-0.0745,0.0000
C01277=89.341,-44.743,13.184,179.7823,-0.3896,0.0000
C01278=87.740,-47.377,13.175,178.9740,-1.5588,0.0000
C01279=86.123,-49.643,13.164,177.4569,-3.2536,0.0000
C01280=84.717,-51.269,13.142,175.1404,-4.9742,0.0000
C01281=83.471,-52.459,13.096,172.2421,-6.9845,0.0000
C01282=82.225,-53.620,13.031,169.6468,-9.9409,0.0000
C01283=80.787,-55.140,12.963,168.0720,-13.2502,0.0000
C01284=78.839,-57.492,12.910,167.3913,-15.6016,0.0000
C01285=76.021,-61.028,12.888,166.7636,-16.1253,0.0000
C01286=72.750,-64.884,12.887,166.0444,-15.5853,0.0000
C01287=68.930,-68.930,12.888,165.2122,-14.7878,0.0000
C01288=64.884,-72.750,12.887,164.4147,-13.9556,0.0000
C01289=61.028,-76.021,12.888,163.8747,-13.2364,0.0000
C01290=57.492,-78.839,12.910,164.3984,-12.6087,0.0000
C01291=55.140,-80.787,12.963,166.7498,-11.9280,0.0000
C01292=53.620,-82.225,13.031,170.0591,-10.3532,0.0000
C01293=52.459,-83.471,13.096,173.0155,-7.7579,0.0000
C01294=51.269,-84.717,13.142,175.0258,-4.8596,0.0000
C01295=49.643,-86.123,13.164,176.7464,-2.5431,0.0000
C01296=47.377,-87.740,13.175,178.4412,-1.0260,0.0000
C01297=44.743,-89.341,13.184,179.6104,-0.2177,0.0000
C01298=42.074,-90.704,13.193,179.9255,-0.0344,0.0000
C01299=39.526,-91.855,13.199,179.9885,-0.0057,0.0000
C01300=37.002,-92.901,13.199,179.9885,-0.0057,0.0000
C01301=34.387,-93.888,13.193,179.9255,-0.0286,0.0000
C01302=31.535,-94.812,13.184,179.5703,-0.1203,0.0000
C01303=28.540,-95.542,13.175,178.1720,-0.3783,0.0000
C01304=25.795,-96.000,13.164,175.9054,-0.5055,0.0000
C01305=23.652,-96.157,13.142,173.0619,-0.0808,0.0000
C01306=21.929,-96.117,13.096,169.6352,0.5534,0.0000
C01307=20.227,-96.057,13.031,165.7998,0.3014,0.0000
C01308=18.135,-96.115,12.963,162.4730,-0.9855,0.0000
C01309=15.094,-96.401,12.910,160.4245,-2.2505,0.0000
C01310=10.602,-96.908,12.888,159.6573,-2.1819,0.0000
C01311=5.562,-97.322,12.887,159.5459,-1.2353,0.0000
C01312=0.000,-97.482,12.888,159.5244,0.0000,0.0000
C01313=0.000,-97.482,12.888,159.5244,0.0000,0.0000
C01314=-5.562,-97.322,12.887,159.5459,1.2353,0.0000
C01315=-10.602,-96.908,12.888,159.6573,2.1819,0.0000
C01316=-15.094,-96.401,12.910,160.4245,2.2505,0.0000
C01317=-18.135,-96.115,12.963,162.4730,0.9855,0.0000
C01318=-20.227,-96.057,13.031,165.7998,-0.3014,0.0000
C01319=-21.929,-96.117,13.096,169.6352,-0.5534,0.0000
C01320=-23.652,-96.157,13.142,173.0619,0.0808,0.0000
C01321=-25.795,-96.000,13.164,175.9054,0.5055,0.0000
C01322=-28.540,-95.542,13.175,178.1720,0.3783,0.0000
C01323=-31.535,-94.812,13.184,179.5703,0.1203,0.0000
C01324=-34.387,-93.888,13.193,179.9255,0.0286,0.0000
C01325=-37.002,-92.901,13.199,179.9885,0.0057,0.0000
C01326=-39.526,-91.855,13.199,179.9885,0.0057,0.0000
C01327=-42.074,-90.704,13.193,179.9255,0.0344,0.0000
C01328=-44.743,-89.341,13.184,179.6104,0.2177,0.0000
C01329=-47.377,-87.740,13.175,178.4412,1.0260,0.0000
C01330=-49.643,-86.123,13.164,176.7464,2.5431,0.0000
C01331=-51.269,-84.717,13.142,175.0258,4.8596,0.0000
C01332=-52.459,-83.471,13.096,173.0155,7.7579,0.0000
C01333=-53.620,-82.225,13.031,170.0591,10.3532,0.0000
C01334=-55.140,-80.787,12.963,166.7498,11.9280,0.0000
C01335=-57.492,-78.839,12.910,164.3984,12.6087,0.0000
C01336=-61.028,-76.021,12.888,163.8747,13.2364,0.0000
C01337=-64.884,-72.750,12.887,164.4147,13.9556,0.0000
C01338=-68.930,-68.930,12.888,165.2122,14.7878,0.0000
C01339=-72.750,-64.884,12.887,166.0444,15.5853,0.0000
C01340=-76.021,-61.028,12.888,166.7636,16.1253,0.0000
C01341=-78.839,-57.492,12.910,167.3913,15.6016,0.0000
C01342=-80.787,-55.140,12.963,168.0720,13.2502,0.0000
C01343=-82.225,-53.620,13.031,169.6468,9.9409,0.0000
C01344=-83.471,-52.459,13.096,172.2421,6.9845,0.0000
C01345=-84.717,-51.269,13.142,175.1404,4.9742,0.0000
C01346=-86.123,-49.643,13.164,177.4569,3.2536,0.0000
C01347=-87.740,-47.377,13.175,178.9740,1.5588,0.0000
C01348=-89.341,-44.743,13.184,179.7823,0.3896,0.0000
C01349=-90.704,-42.074,13.193,179.9656,0.0745,0.0000
C01350=-91.855,-39.526,13.199,179.9943,0.0115,0.0000
C01351=-92.901,-37.002,13.199,179.9943,0.0115,0.0000
C01352=-93.888,-34.387,13.193,179.9714,0.0745,0.0000
C01353=-94.812,-31.535,13.184,179.8797,0.4297,0.0000
C01354=-95.542,-28.540,13.175,179.6217,1.8280,0.0000
C01355=-96.000,-25.795,13.164,179.4945,4.0946,0.0000
C01356=-96.157,-23.652,13.142,179.9192,6.9381,0.0000
C01357=-96.117,-21.929,13.096,-179.4466,10.3648,0.0000
C01358=-96.057,-20.227,13.031,-179.6986,14.2002,0.0000
C01359=-96.115,-18.135,12.963,179.0145,17.5270,0.0000
C01360=-96.401,-15.094,12.910,177.7495,19.5755,0.0000
C01361=-96.908,-10.602,12.888,177.8181,20.3427,0.0000
C01362=-97.322,-5.562,12.887,178.7647,20.4541,0.0000
C01363=-97.482,0.000,12.888,-180.0000,20.4756,0.0000
C01364=-97.322,5.562,12.887,-178.7647,20.4541,0.0000
C01365=-96.908,10.602,12.888,-177.8181,20.3427,0.0000
C01366=-96.401,15.094,12.910,-177.7495,19.5755,0.0000
C01367=-96.115,18.135,12.963,-179.0145,17.5270,0.0000
C01368=-96.057,20.227,13.031,179.6986,14.2002,0.0000
C01369=-96.117,21.929,13.096,179.4466,10.3648,0.0000
C01370=-96.157,23.652,13.142,-179.9192,6.9381,0.0000
C01371=-96.000,25.795,13.164,-179.4945,4.0946,0.0000
C01372=-95.542,28.540,13.175,-179.6217,1.8280,0.0000
C01373=-94.812,31.535,13.184,-179.8797,0.4297,0.0000
C01374=-93.888,34.387,13.193,-179.9714,0.0745,0.0000
C01375=-92.901,37.002,13.199,-179.9943,0.0115,0.0000
C01376=-91.855,39.526,13.199,-179.9943,0.0115,0.0000
C01377=-90.704,42.074,13.193,-179.9656,0.0745,0.0000
C01378=-89.341,44.743,13.184,-179.7823,0.3896,0.0000
C01379=-87.740,47.377,13.175,-178.9740,1.5588,0.0000
C01380=-86.123,49.643,13.164,-177.4569,3.2536,0.0000
C01381=-84.717,51.269,13.142,-175.1404,4.9742,0.0000
C01382=-83.471,52.459,13.096,-172.2421,6.9845,0.0000
C01383=-82.225,53.620,13.031,-169.6468,9.9409,0.0000
C01384=-80.787,55.140,12.963,-168.0720,13.2502,0.0000
C01385=-78.839,57.492,12.910,-167.3913,15.6016,0.0000
C01386=-76.021,61.028,12.888,-166.7636,16.1253,0.0000
C01387=-72.750,64.884,12.887,-166.0444,15.5853,0.0000
C01388=-68.930,68.930,12.888,-165.2122,14.7878,0.0000
C01389=-64.884,72.750,12.887,-164.4147,13.9556,0.0000
C01390=-61.028,76.021,12.888,-163.8747,13.2364,0.0000
C01391=-57.492,78.839,12.910,-164.3984,12.6087,0.0000
C01392=-55.140,80.787,12.963,-166.7498,11.9280,0.0000
C01393=-53.620,82.225,13.031,-170.0591,10.3532,0.0000
C01394=-52.459,83.471,13.096,-173.0155,7.7579,0.0000
C01395=-51.269,84.717,13.142,-175.0258,4.8596,0.0000
C01396=-49.643,86.123,13.164,-176.7464,2.5431,0.0000
C01397=-47.377,87.740,13.175,-178.4412,1.0260,0.0000
C01398=-44.743,89.341,13.184,-179.6104,0.2177,0.0000
C01399=-42.074,90.704,13.193,-179.9255,0.0344,0.0000
C01400=-39.526,91.855,13.199,-179.9885,0.0057,0.0000
C01401=-37.002,92.901,13.199,-179.9885,0.0057,0.0000
C01402=-34.387,93.888,13.193,-179.9255,0.0286,0.0000
C01403=-31.535,94.812,13.184,-179.5703,0.1203,0.0000
C01404=-28.540,95.542,13.175,-178.1720,0.3783,0.0000
C01405=-25.795,96.000,13.164,-175.9054,0.5055,0.0000
C01406=-23.652,96.157,13.142,-173.0619,0.0808,0.0000
C01407=-21.929,96.117,13.096,-169.6352,-0.5534,0.0000
C01408=-20.227,96.057,13.031,-165.7998,-0.3014,0.0000
C01409=-18.135,96.115,12.963,-162.4730,0.9855,0.0000
C01410=-15.094,96.401,12.910,-160.4245,2.2505,0.0000
C01411=-10.602,96.908,12.888,-159.6573,2.1819,0.0000
C01412=-5.562,97.322,12.887,-159.5459,1.2353,0.0000
C01413=0.000,97.482,12.888,-159.5244,0.0000,0.0000
C01414=0.000,96.668,14.931,-157.0813,0.0000,0.0000
C01415=5.488,96.511,14.930,-157.1024,-1.3932,0.0000
C01416=10.476,96.104,14.932,-157.2253,-2.4116,0.0000
C01417=14.942,95.628,14.964,-158.0602,-2.1869,0.0000
C01418=17.951,95.422,15.043,-160.4761,-0.1520,0.0000
C01419=20.020,95.481,15.144,-164.5735,1.5931,0.0000
C01420=21.708,95.685,15.242,-169.0723,1.6632,0.0000
C01421=23.417,95.878,15.312,-172.7037,0.5199,0.0000
C01422=25.541,95.862,15.345,-175.6699,-0.3103,0.0000
C01423=28.302,95.513,15.362,-178.1088,-0.3268,0.0000
C01424=31.347,94.846,15.376,-179.5932,-0.1089,0.0000
C01425=34.268,93.927,15.390,-179.9198,-0.0286,0.0000
C01426=36.962,92.916,15.399,-179.9885,-0.0057,0.0000
C01427=39.566,91.838,15.399,-179.9885,-0.0057,0.0000
C01428=42.186,90.648,15.390,-179.9255,-0.0344,0.0000
C01429=44.901,89.232,15.376,-179.6390,-0.2120,0.0000
C01430=47.525,87.551,15.362,-178.4295,-1.1063,0.0000
C01431=49.724,85.845,15.345,-176.7167,-2.8478,0.0000
C01432=51.237,84.354,15.312,-175.1938,-5.5338,0.0000
C01433=52.309,83.010,15.242,-173.3806,-8.9229,0.0000
C01434=53.359,81.672,15.144,-170.0466,-12.1240,0.0000
C01435=54.780,80.167,15.043,-165.8222,-13.9719,0.0000
C01436=57.054,78.185,14.964,-162.6791,-14.4572,0.0000
C01437=60.548,75.364,14.932,-161.9128,-14.9558,0.0000
C01438=64.363,72.124,14.930,-162.4712,-15.7184,0.0000
C01439=68.355,68.355,14.931,-163.3521,-16.6479,0.0000
C01440=72.124,64.363,14.930,-164.2816,-17.5288,0.0000
C01441=75.364,60.548,14.932,-165.0442,-18.0872,0.0000
C01442=78.185,57.054,14.964,-165.5428,-17.3209,0.0000
C01443=80.167,54.780,15.043,-166.0281,-14.1778,0.0000
C01444=81.672,53.359,15.144,-167.8760,-9.9534,0.0000
C01445=83.010,52.309,15.242,-171.0771,-6.6194,0.0000
C01446=84.354,51.237,15.312,-174.4662,-4.8062,0.0000
C01447=85.845,49.724,15.345,-177.1522,-3.2833,0.0000
C01448=87.551,47.525,15.362,-178.8937,-1.5705,0.0000
C01449=89.232,44.901,15.376,-179.7880,-0.3610,0.0000
C01450=90.648,42.186,15.390,-179.9656,-0.0745,0.0000
C01451=91.838,39.566,15.399,-179.9943,-0.0115,0.0000
C01452=92.916,36.962,15.399,-179.9943,-0.0115,0.0000
C01453=93.927,34.268,15.390,-179.9714,-0.0802,0.0000
C01454=94.846,31.347,15.376,-179.8911,-0.4068,0.0000
C01455=95.513,28.302,15.362,-179.6732,-1.8912,0.0000
C01456=95.862,25.541,15.345,-179.6897,-4.3301,0.0000
C01457=95.878,23.417,15.312,179.4801,-7.2963,0.0000
C01458=95.685,21.708,15.242,178.3368,-10.9277,0.0000
C01459=95.481,20.020,15.144,178.4069,-15.4265,0.0000
C01460=95.422,17.951,15.043,-179.8480,-19.5239,0.0000
C01461=95.628,14.942,14.964,-177.8131,-21.9398,0.0000
C01462=96.104,10.476,14.932,-177.5884,-22.7747,0.0000
C01463=96.511,5.488,14.930,-178.6068,-22.8976,0.0000
C01464=96.668,0.000,14.931,180.0000,-22.9187,0.0000
C01465=96.511,-5.488,14.930,178.6068,-22.8976,0.0000
C01466=96.104,-10.476,14.932,177.5884,-22.7747,0.0000
C01467=95.628,-14.942,14.964,177.8131,-21.9398,0.0000
C01468=95.422,-17.951,15.043,179.8480,-19.5239,0.0000
C01469=95.481,-20.020,15.144,-178.4069,-15.4265,0.0000
C01470=95.685,-21.708,15.242,-178.3368,-10.9277,0.0000
C01471=95.878,-23.417,15.312,-179.4801,-7.2963,0.0000
C01472=95.862,-25.541,15.345,179.6897,-4.3301,0.0000
C01473=95.513,-28.302,15.362,179.6732,-1.8912,0.0000
C01474=94.846,-31.347,15.376,179.8911,-0.4068,0.0000
C01475=93.927,-34.268,15.390,179.9714,-0.0802,0.0000
C01476=92.916,-36.962,15.399,179.9943,-0.0115,0.0000
C01477=91.838,-39.566,15.399,179.9943,-0.0115,0.0000
C01478=90.648,-42.186,15.390,179.9656,-0.0745,0.0000
C01479=89.232,-44.901,15.376,179.7880,-0.3610,0.0000
C01480=87.551,-47.525,15.362,178.8937,-1.5705,0.0000
C01481=85.845,-49.724,15.345,177.1522,-3.2833,0.0000
C01482=84.354,-51.237,15.312,174.4662,-4.8062,0.0000
C01483=83.010,-52.309,15.242,171.0771,-6.6194,0.0000
C01484=81.672,-53.359,15.144,167.8760,-9.9534,0.0000
C01485=80.167,-54.780,15.043,166.0281,-14.1778,0.0000
C01486=78.185,-57.054,14.964,165.5428,-17.3209,0.0000
C01487=75.364,-60.548,14.932,165.0442,-18.0872,0.0000
C01488=72.124,-64.363,14.930,164.2816,-17.5288,0.0000
C01489=68.355,-68.355,14.931,163.3521,-16.6479,0.0000
C01490=64.363,-72.124,14.930,162.4712,-15.7184,0.0000
C01491=60.548,-75.364,14.932,161.9128,-14.9558,0.0000
C01492=57.054,-78.185,14.964,162.6791,-14.4572,0.0000
C01493=54.780,-80.167,15.043,165.8222,-13.9719,0.0000
C01494=53.359,-81.672,15.144,170.0466,-12.1240,0.0000
C01495=52.309,-83.010,15.242,173.3806,-8.9229,0.0000
C01496=51.237,-84.354,15.312,175.1938,-5.5338,0.0000
C01497=49.724,-85.845,15.345,176.7167,-2.8478,0.0000
C01498=47.525,-87.551,15.362,178.4295,-1.1063,0.0000
C01499=44.901,-89.232,15.376,179.6390,-0.2120,0.0000
C01500=42.186,-90.648,15.390,179.9255,-0.0344,0.0000
C01501=39.566,-91.838,15.399,179.9885,-0.0057,0.0000
C01502=36.962,-92.916,15.399,179.9885,-0.0057,0.0000
C01503=34.268,-93.927,15.390,179.9198,-0.0286,0.0000
C01504=31.347,-94.846,15.376,179.5932,-0.1089,0.0000
C01505=28.302,-95.513,15.362,178.1088,-0.3268,0.0000
C01506=25.541,-95.862,15.345,175.6699,-0.3103,0.0000
C01507=23.417,-95.878,15.312,172.7037,0.5199,0.0000
C01508=21.708,-95.685,15.242,169.0723,1.6632,0.0000
C01509=20.020,-95.481,15.144,164.5735,1.5931,0.0000
C01510=17.951,-95.422,15.043,160.4761,-0.1520,0.0000
C01511=14.942,-95.628,14.964,158.0602,-2.1869,0.0000
C01512=10.476,-96.104,14.932,157.2253,-2.4116,0.0000
C01513=5.488,-96.511,14.930,157.1024,-1.3932,0.0000
C01514=0.000,-96.668,14.931,157.0813,0.0000,0.0000
C01515=0.000,-96.668,14.931,157.0813,0.0000,0.0000
C01516=-5.488,-96.511,14.930,157.1024,1.3932,0.0000
C01517=-10.476,-96.104,14.932,157.2253,2.4116,0.0000
C01518=-14.942,-95.628,14.964,158.0602,2.1869,0.0000
C01519=-17.951,-95.422,15.043,160.4761,0.1520,0.0000
C01520=-20.020,-95.481,15.144,164.5735,-1.5931,0.0000
C01521=-21.708,-95.685,15.242,169.0723,-1.6632,0.0000
C01522=-23.417,-95.878,15.312,172.7037,-0.5199,0.0000
C01523=-25.541,-95.862,15.345,175.6699,0.3103,0.0000
C01524=-28.302,-95.513,15.362,178.1088,0.3268,0.0000
C01525=-31.347,-94.846,15.376,179.5932,0.1089,0.0000
C01526=-34.268,-93.927,15.390,179.9198,0.0286,0.0000
C01527=-36.962,-92.916,15.399,179.9885,0.0057,0.0000
C01528=-39.566,-91.838,15.399,179.9885,0.0057,0.0000
C01529=-42.186,-90.648,15.390,179.9255,0.0344,0.0000
C01530=-44.901,-89.232,15.376,179.6390,0.2120,0.0000
C01531=-47.525,-87.551,15.362,178.4295,1.1063,0.0000
C01532=-49.724,-85.845,15.345,176.7167,2.8478,0.0000
C01533=-51.237,-84.354,15.312,175.1938,5.5338,0.0000
C01534=-52.309,-83.010,15.242,173.3806,8.9229,0.0000
C01535=-53.359,-81.672,15.144,170.0466,12.1240,0.0000
C01536=-54.780,-80.167,15.043,165.8222,13.9719,0.0000
C01537=-57.054,-78.185,14.964,162.6791,14.4572,0.0000
C01538=-60.548,-75.364,14.932,161.9128,14.9558,0.0000
C01539=-64.363,-72.124,14.930,162.4712,15.7184,0.0000
C01540=-68.355,-68.355,14.931,163.3521,16.6479,0.0000
C01541=-72.124,-64.363,14.930,164.2816,17.5288,0.0000
C01542=-75.364,-60.548,14.932,165.0442,18.0872,0.0000
C01543=-78.185,-57.054,14.964,165.5428,17.3209,0.0000
C01544=-80.167,-54.780,15.043,166.0281,14.1778,0.0000
C01545=-81.672,-53.359,15.144,167.8760,9.9534,0.0000
C01546=-83.010,-52.309,15.242,171.0771,6.6194,0.0000
C01547=-84.354,-51.237,15.312,174.4662,4.8062,0.0000
C01548=-85.845,-49.724,15.345,177.1522,3.2833,0.0000
C01549=-87.551,-47.525,15.362,178.8937,1.5705,0.0000
C01550=-89.232,-44.901,15.376,179.7880,0.3610,0.0000
C01551=-90.648,-42.186,15.390,179.9656,0.0745,0.0000
C01552=-91.838,-39.566,15.399,179.9943,0.0115,0.0000
C01553=-92.916,-36.962,15.399,179.9943,0.0115,0.0000
C01554=-93.927,-34.268,15.390,179.9714,0.0802,0.0000
C01555=-94.846,-31.347,15.376,179.8911,0.4068,0.0000
C01556=-95.513,-28.302,15.362,179.6732,1.8912,0.0000
C01557=-95.862,-25.541,15.345,179.6897,4.3301,0.0000
C01558=-95.878,-23.417,15.312,-179.4801,7.2963,0.0000
C01559=-95.685,-21.708,15.242,-178.3368,10.9277,0.0000
C01560=-95.481,-20.020,15.144,-178.4069,15.4265,0.0000
C01561=-95.422,-17.951,15.043,179.8480,19.5239,0.0000
C01562=-95.628,-14.942,14.964,177.8131,21.9398,0.0000
C01563=-96.104,-10.476,14.932,177.5884,22.7747,0.0000
C01564=-96.511,-5.488,14.930,178.6068,22.8976,0.0000
C01565=-96.668,0.000,14.931,-180.0000,22.9187,0.0000
C01566=-96.511,5.488,14.930,-178.6068,22.8976,0.0000
C01567=-96.104,10.476,14.932,-177.5884,22.7747,0.0000
C01568=-95.628,14.942,14.964,-177.8131,21.9398,0.0000
C01569=-95.422,17.951,15.043,-179.8480,19.5239,0.0000
C01570=-95.481,20.020,15.144,178.4069,15.4265,0.0000
C01571=-95.685,21.708,15.242,178.3368,10.9277,0.0000
C01572=-95.878,23.417,15.312,179.4801,7.2963,0.0000
C01573=-95.862,25.541,15.345,-179.6897,4.3301,0.0000
C01574=-95.513,28.302,15.362,-179.6732,1.8912,0.0000
C01575=-94.846,31.347,15.376,-179.8911,0.4068,0.0000
C01576=-93.927,34.268,15.390,-179.9714,0.0802,0.0000
C01577=-92.916,36.962,15.399,-179.9943,0.0115,0.0000
C01578=-91.838,39.566,15.399,-179.9943,0.0115,0.0000
C01579=-90.648,42.186,15.390,-179.9656,0.0745,0.0000
C01580=-89.232,44.901,15.376,-179.7880,0.3610,0.0000
C01581=-87.551,47.525,15.362,-178.8937,1.5705,0.0000
C01582=-85.845,49.724,15.345,-177.1522,3.2833,0.0000
C01583=-84.354,51.237,15.312,-174.4662,4.8062,0.0000
C01584=-83.010,52.309,15.242,-171.0771,6.6194,0.0000
C01585=-81.672,53.359,15.144,-167.8760,9.9534,0.0000
C01586=-80.167,54.780,15.043,-166.0281,14.1778,0.0000
C01587=-78.185,57.054,14.964,-165.5428,17.3209,0.0000
C01588=-75.364,60.548,14.932,-165.0442,18.0872,0.0000
C01589=-72.124,64.363,14.930,-164.2816,17.5288,0.0000
C01590=-68.355,68.355,14.931,-163.3521,16.6479,0.0000
C01591=-64.363,72.124,14.930,-162.4712,15.7184,0.0000
C01592=-60.548,75.364,14.932,-161.9128,14.9558,0.0000
C01593=-57.054,78.185,14.964,-162.6791,14.4572,0.0000
C01594=-54.780,80.167,15.043,-165.8222,13.9719,0.0000
C01595=-53.359,81.672,15.144,-170.0466,12.1240,0.0000
C01596=-52.309,83.010,15.242,-173.3806,8.9229,0.0000
C01597=-51.237,84.354,15.312,-175.1938,5.5338,0.0000
C01598=-49.724,85.845,15.345,-176.7167,2.8478,0.0000
C01599=-47.525,87.551,15.362,-178.4295,1.1063,0.0000
C01600=-44.901,89.232,15.376,-179.6390,0.2120,0.0000
C01601=-42.186,90.648,15.390,-179.9255,0.0344,0.0000
C01602=-39.566,91.838,15.399,-179.9885,0.0057,0.0000
C01603=-36.962,92.916,15.399,-179.9885,0.0057,0.0000
C01604=-34.268,93.927,15.390,-179.9198,0.0286,0.0000
C01605=-31.347,94.846,15.376,-179.5932,0.1089,0.0000
C01606=-28.302,95.513,15.362,-178.1088,0.3268,0.0000
C01607=-25.541,95.862,15.345,-175.6699,0.3103,0.0000
C01608=-23.417,95.878,15.312,-172.7037,-0.5199,0.0000
C01609=-21.708,95.685,15.242,-169.0723,-1.6632,0.0000
C01610=-20.020,95.481,15.144,-164.5735,-1.5931,0.0000
C01611=-17.951,95.422,15.043,-160.4761,0.1520,0.0000
C01612=-14.942,95.628,14.964,-158.0602,2.1869,0.0000
C01613=-10.476,96.104,14.932,-157.2253,2.4116,0.0000
C01614=-5.488,96.511,14.930,-157.1024,1.3932,0.0000
C01615=0.000,96.668,14.931,-157.0813,0.0000,0.0000
C01616=0.000,95.772,16.941,-154.8879,0.0000,0.0000
C01617=5.406,95.617,16.939,-154.9114,-1.5437,0.0000
C01618=10.339,95.219,16.941,-155.0354,-2.5917,0.0000
C01619=14.774,94.777,16.986,-155.9403,-1.9704,0.0000
C01620=17.748,94.656,17.095,-158.8477,1.0076,0.0000
C01621=19.790,94.842,17.237,-163.9080,3.1497,0.0000
C01622=21.462,95.203,17.374,-169.0805,2.8662,0.0000
C01623=23.155,95.565,17.473,-172.7371,1.2014,0.0000
C01624=25.257,95.708,17.521,-175.6241,-0.0575,0.0000
C01625=28.035,95.481,17.545,-178.1262,-0.2580,0.0000
C01626=31.135,94.884,17.565,-179.6505,-0.0859,0.0000
C01627=34.135,93.972,17.585,-179.9255,-0.0286,0.0000
C01628=36.917,92.934,17.598,-179.9943,-0.0057,0.0000
C01629=39.610,91.818,17.598,-179.9943,-0.0057,0.0000
C01630=42.311,90.585,17.585,-179.9255,-0.0344,0.0000
C01631=45.077,89.109,17.565,-179.6906,-0.1891,0.0000
C01632=47.692,87.339,17.545,-178.4927,-1.1406,0.0000
C01633=49.816,85.535,17.521,-176.8600,-3.0598,0.0000
C01634=51.202,83.948,17.473,-175.6928,-5.9919,0.0000
C01635=52.143,82.495,17.374,-174.2298,-9.7548,0.0000
C01636=53.070,81.058,17.237,-170.6258,-13.6548,0.0000
C01637=54.382,79.482,17.095,-165.3654,-15.9665,0.0000
C01638=56.571,77.464,16.986,-161.2174,-16.2426,0.0000
C01639=60.019,74.640,16.941,-160.1389,-16.5517,0.0000
C01640=63.789,71.434,16.939,-160.7038,-17.3288,0.0000
C01641=67.721,67.721,16.941,-161.6638,-18.3362,0.0000
C01642=71.434,63.789,16.939,-162.6712,-19.2962,0.0000
C01643=74.640,60.019,16.941,-163.4483,-19.8611,0.0000
C01644=77.464,56.571,16.986,-163.7574,-18.7826,0.0000
C01645=79.482,54.382,17.095,-164.0335,-14.6346,0.0000
C01646=81.058,53.070,17.237,-166.3452,-9.3742,0.0000
C01647=82.495,52.143,17.374,-170.2452,-5.7702,0.0000
C01648=83.948,51.202,17.473,-174.0081,-4.3072,0.0000
C01649=85.535,49.816,17.521,-176.9402,-3.1400,0.0000
C01650=87.339,47.692,17.545,-178.8594,-1.5073,0.0000
C01651=89.109,45.077,17.565,-179.8109,-0.3094,0.0000
C01652=90.585,42.311,17.585,-179.9656,-0.0745,0.0000
C01653=91.818,39.610,17.598,-179.9943,-0.0057,0.0000
C01654=92.934,36.917,17.598,-179.9943,-0.0057,0.0000
C01655=93.972,34.135,17.585,-179.9714,-0.0745,0.0000
C01656=94.884,31.135,17.565,-179.9141,-0.3495,0.0000
C01657=95.481,28.035,17.545,-179.7420,-1.8738,0.0000
C01658=95.708,25.257,17.521,-179.9425,-4.3759,0.0000
C01659=95.565,23.155,17.473,178.7986,-7.2629,0.0000
C01660=95.203,21.462,17.374,177.1338,-10.9195,0.0000
C01661=94.842,19.790,17.237,176.8503,-16.0920,0.0000
C01662=94.656,17.748,17.095,178.9924,-21.1523,0.0000
C01663=94.777,14.774,16.986,-178.0296,-24.0597,0.0000
C01664=95.219,10.339,16.941,-177.4083,-24.9646,0.0000
C01665=95.617,5.406,16.939,-178.4563,-25.0886,0.0000
C01666=95.772,0.000,16.941,180.0000,-25.1121,0.0000
C01667=95.617,-5.406,16.939,178.4563,-25.0886,0.0000
C01668=95.219,-10.339,16.941,177.4083,-24.9646,0.0000
C01669=94.777,-14.774,16.986,178.0233,-24.0597,0.0000
C01670=94.656,-17.748,17.095,-178.9924,-21.1523,0.0000
C01671=94.842,-19.790,17.237,-176.8503,-16.0920,0.0000
C01672=95.203,-21.462,17.374,-177.1338,-10.9195,0.0000
C01673=95.565,-23.155,17.473,-178.7986,-7.2629,0.0000
C01674=95.708,-25.257,17.521,179.9425,-4.3759,0.0000
C01675=95.481,-28.035,17.545,179.7420,-1.8738,0.0000
C01676=94.884,-31.135,17.565,179.9141,-0.3495,0.0000
C01677=93.972,-34.135,17.585,179.9714,-0.0745,0.0000
C01678=92.934,-36.917,17.598,179.9943,-0.0057,0.0000
C01679=91.818,-39.610,17.598,179.9943,-0.0057,0.0000
C01680=90.585,-42.311,17.585,179.9656,-0.0745,0.0000
C01681=89.109,-45.077,17.565,179.8109,-0.3094,0.0000
C01682=87.339,-47.692,17.545,178.8594,-1.5073,0.0000
C01683=85.535,-49.816,17.521,176.9402,-3.1400,0.0000
C01684=83.948,-51.202,17.473,174.0081,-4.3072,0.0000
C01685=82.495,-52.143,17.374,170.2452,-5.7702,0.0000
C01686=81.058,-53.070,17.237,166.3452,-9.3742,0.0000
C01687=79.482,-54.382,17.095,164.0335,-14.6346,0.0000
C01688=77.464,-56.571,16.986,163.7574,-18.7826,0.0000
C01689=74.640,-60.019,16.941,163.4483,-19.8611,0.0000
C01690=71.434,-63.789,16.939,162.6712,-19.2962,0.0000
C01691=67.721,-67.721,16.941,161.6638,-18.3362,0.0000
C01692=63.789,-71.434,16.939,160.7038,-17.3288,0.0000
C01693=60.019,-74.640,16.941,160.1389,-16.5517,0.0000
C01694=56.571,-77.464,16.986,161.2174,-16.2426,0.0000
C01695=54.382,-79.482,17.095,165.3654,-15.9665,0.0000
C01696=53.070,-81.058,17.237,170.6258,-13.6548,0.0000
C01697=52.143,-82.495,17.374,174.2298,-9.7548,0.0000
C01698=51.202,-83.948,17.473,175.6928,-5.9919,0.0000
C01699=49.816,-85.535,17.521,176.8600,-3.0598,0.0000
C01700=47.692,-87.339,17.545,178.4927,-1.1406,0.0000
C01701=45.077,-89.109,17.565,179.6906,-0.1891,0.0000
C01702=42.311,-90.585,17.585,179.9255,-0.0344,0.0000
C01703=39.610,-91.818,17.598,179.9943,-0.0057,0.0000
C01704=36.917,-92.934,17.598,179.9943,-0.0057,0.0000
C01705=34.135,-93.972,17.585,179.9255,-0.0286,0.0000
C01706=31.135,-94.884,17.565,179.6505,-0.0859,0.0000
C01707=28.035,-95.481,17.545,178.1262,-0.2580,0.0000
C01708=25.257,-95.708,17.521,175.6241,-0.0575,0.0000
C01709=23.155,-95.565,17.473,172.7371,1.2014,0.0000
C01710=21.462,-95.203,17.374,169.0805,2.8662,0.0000
C01711=19.790,-94.842,17.237,163.9080,3.1497,0.0000
C01712=17.748,-94.656,17.095,158.8477,1.0076,0.0000
C01713=14.774,-94.777,16.986,155.9403,-1.9704,0.0000
C01714=10.339,-95.219,16.941,155.0354,-2.5917,0.0000
C01715=5.406,-95.617,16.939,154.9114,-1.5437,0.0000
C01716=0.000,-95.772,16.941,154.8879,0.0000,0.0000
C01717=0.000,-95.772,16.941,154.8879,0.0000,0.0000
C01718=-5.406,-95.617,16.939,154.9114,1.5437,0.0000
C01719=-10.339,-95.219,16.941,155.0354,2.5917,0.0000
C01720=-14.774,-94.777,16.986,155.9403,1.9767,0.0000
C01721=-17.748,-94.656,17.095,158.8477,-1.0076,0.0000
C01722=-19.790,-94.842,17.237,163.9080,-3.1497,0.0000
C01723=-21.462,-95.203,17.374,169.0805,-2.8662,0.0000
C01724=-23.155,-95.565,17.473,172.7371,-1.2014,0.0000
C01725=-25.257,-95.708,17.521,175.6241,0.0575,0.0000
C01726=-28.035,-95.481,17.545,178.1262,0.2580,0.0000
C01727=-31.135,-94.884,17.565,179.6505,0.0859,0.0000
C01728=-34.135,-93.972,17.585,179.9255,0.0286,0.0000
C01729=-36.917,-92.934,17.598,179.9943,0.0057,0.0000
C01730=-39.610,-91.818,17.598,179.9943,0.0057,0.0000
C01731=-42.311,-90.585,17.585,179.9255,0.0344,0.0000
C01732=-45.077,-89.109,17.565,179.6906,0.1891,0.0000
C01733=-47.692,-87.339,17.545,178.4927,1.1406,0.0000
C01734=-49.816,-85.535,17.521,176.8600,3.0598,0.0000
C01735=-51.202,-83.948,17.473,175.6928,5.9919,0.0000
C01736=-52.143,-82.495,17.374,174.2298,9.7548,0.0000
C01737=-53.070,-81.058,17.237,170.6258,13.6548,0.0000
C01738=-54.382,-79.482,17.095,165.3654,15.9665,0.0000
C01739=-56.571,-77.464,16.986,161.2174,16.2426,0.0000
C01740=-60.019,-74.640,16.941,160.1389,16.5517,0.0000
C01741=-63.789,-71.434,16.939,160.7038,17.3288,0.0000
C01742=-67.721,-67.721,16.941,161.6638,18.3362,0.0000
C01743=-71.434,-63.789,16.939,162.6712,19.2962,0.0000
C01744=-74.640,-60.019,16.941,163.4483,19.8611,0.0000
C01745=-77.464,-56.571,16.986,163.7574,18.7826,0.0000
C01746=-79.482,-54.382,17.095,164.0335,14.6346,0.0000
C01747=-81.058,-53.070,17.237,166.3452,9.3742,0.0000
C01748=-82.495,-52.143,17.374,170.2452,5.7702,0.0000
C01749=-83.948,-51.202,17.473,174.0081,4.3072,0.0000
C01750=-85.535,-49.816,17.521,176.9402,3.1400,0.0000
C01751=-87.339,-47.692,17.545,178.8594,1.5073,0.0000
C01752=-89.109,-45.077,17.565,179.8109,0.3094,0.0000
C01753=-90.585,-42.311,17.585,179.9656,0.0745,0.0000
C01754=-91.818,-39.610,17.598,179.9943,0.0057,0.0000
C01755=-92.934,-36.917,17.598,179.9943,0.0057,0.0000
C01756=-93.972,-34.135,17.585,179.9714,0.0745,0.0000
C01757=-94.884,-31.135,17.565,179.9141,0.3495,0.0000
C01758=-95.481,-28.035,17.545,179.7420,1.8738,0.0000
C01759=-95.708,-25.257,17.521,179.9425,4.3759,0.0000
C01760=-95.565,-23.155,17.473,-178.7986,7.2629,0.0000
C01761=-95.203,-21.462,17.374,-177.1338,10.9195,0.0000
C01762=-94.842,-19.790,17.237,-176.8503,16.0920,0.0000
C01763=-94.656,-17.748,17.095,-178.9924,21.1523,0.0000
C01764=-94.777,-14.774,16.986,178.0296,24.0597,0.0000
C01765=-95.219,-10.339,16.941,177.4083,24.9646,0.0000
C01766=-95.617,-5.406,16.939,178.4563,25.0886,0.0000
C01767=-95.772,0.000,16.941,-180.0000,25.1121,0.0000
C01768=-95.617,5.406,16.939,-178.4563,25.0886,0.0000
C01769=-95.219,10.339,16.941,-177.4083,24.9646,0.0000
C01770=-94.777,14.774,16.986,-178.0233,24.0597,0.0000
C01771=-94.656,17.748,17.095,178.9924,21.1523,0.0000
C01772=-94.842,19.790,17.237,176.8503,16.0920,0.0000
C01773=-95.203,21.462,17.374,177.1338,10.9195,0.0000
C01774=-95.565,23.155,17.473,178.7986,7.2629,0.0000
C01775=-95.708,25.257,17.521,-179.9425,4.3759,0.0000
C01776=-95.481,28.035,17.545,-179.7420,1.8738,0.0000
C01777=-94.884,31.135,17.565,-179.9141,0.3495,0.0000
C01778=-93.972,34.135,17.585,-179.9714,0.0745,0.0000
C01779=-92.934,36.917,17.598,-179.9943,0.0057,0.0000
C01780=-91.818,39.610,17.598,-179.9943,0.0057,0.0000
C01781=-90.585,42.311,17.585,-179.9656,0.0745,0.0000
C01782=-89.109,45.077,17.565,-179.8109,0.3094,0.0000
C01783=-87.339,47.692,17.545,-178.8594,1.5073,0.0000
C01784=-85.535,49.816,17.521,-176.9402,3.1400,0.0000
C01785=-83.948,51.202,17.473,-174.0081,4.3072,0.0000
C01786=-82.495,52.143,17.374,-170.2452,5.7702,0.0000
C01787=-81.058,53.070,17.237,-166.3452,9.3742,0.0000
C01788=-79.482,54.382,17.095,-164.0335,14.6346,0.0000
C01789=-77.464,56.571,16.986,-163.7574,18.7826,0.0000
C01790=-74.640,60.019,16.941,-163.4483,19.8611,0.0000
C01791=-71.434,63.789,16.939,-162.6712,19.2962,0.0000
C01792=-67.721,67.721,16.941,-161.6638,18.3362,0.0000
C01793=-63.789,71.434,16.939,-160.7038,17.3288,0.0000
C01794=-60.019,74.640,16.941,-160.1389,16.5517,0.0000
C01795=-56.571,77.464,16.986,-161.2174,16.2426,0.0000
C01796=-54.382,79.482,17.095,-165.3654,15.9665,0.0000
C01797=-53.070,81.058,17.237,-170.6258,13.6548,0.0000
C01798=-52.143,82.495,17.374,-174.2298,9.7548,0.0000
C01799=-51.202,83.948,17.473,-175.6928,5.9919,0.0000
C01800=-49.816,85.535,17.521,-176.8600,3.0598,0.0000
C01801=-47.692,87.339,17.545,-178.4927,1.1406,0.0000
C01802=-45.077,89.109,17.565,-179.6906,0.1891,0.0000
C01803=-42.311,90.585,17.585,-179.9255,0.0344,0.0000
C01804=-39.610,91.818,17.598,-179.9943,0.0057,0.0000
C01805=-36.917,92.934,17.598,-179.9943,0.0057,0.0000
C01806=-34.135,93.972,17.585,-179.9255,0.0286,0.0000
C01807=-31.135,94.884,17.565,-179.6505,0.0859,0.0000
C01808=-28.035,95.481,17.545,-178.1262,0.2580,0.0000
C01809=-25.257,95.708,17.521,-175.6241,0.0575,0.0000
C01810=-23.155,95.565,17.473,-172.7371,-1.2014,0.0000
C01811=-21.462,95.203,17.374,-169.0805,-2.8662,0.0000
C01812=-19.790,94.842,17.237,-163.9080,-3.1497,0.0000
C01813=-17.748,94.656,17.095,-158.8477,-1.0076,0.0000
C01814=-14.774,94.777,16.986,-155.9403,1.9767,0.0000
C01815=-10.339,95.219,16.941,-155.0354,2.5917,0.0000
C01816=-5.406,95.617,16.939,-154.9114,1.5437,0.0000
C01817=0.000,95.772,16.941,-154.8879,0.0000,0.0000
C01818=0.000,94.804,18.916,-152.9225,0.0000,0.0000
C01819=5.317,94.652,18.914,-152.9505,-1.6728,0.0000
C01820=10.190,94.262,18.917,-153.0810,-2.7315,0.0000
C01821=14.592,93.857,18.976,-154.0604,-1.6120,0.0000
C01822=17.528,93.824,19.120,-157.6161,2.4729,0.0000
C01823=19.540,94.146,19.309,-163.8596,4.8117,0.0000
C01824=21.192,94.676,19.493,-169.6643,3.9748,0.0000
C01825=22.867,95.222,19.627,-173.1679,1.8469,0.0000
C01826=24.945,95.538,19.692,-175.7793,0.2183,0.0000
C01827=27.741,95.446,19.726,-178.2350,-0.1777,0.0000
C01828=30.903,94.927,19.753,-179.7307,-0.0630,0.0000
C01829=33.988,94.020,19.780,-179.9255,-0.0229,0.0000
C01830=36.867,92.953,19.798,-179.9943,-0.0057,0.0000
C01831=39.659,91.796,19.798,-179.9943,-0.0057,0.0000
C01832=42.449,90.515,19.780,-179.9312,-0.0344,0.0000
C01833=45.272,88.975,19.753,-179.7708,-0.1490,0.0000
C01834=47.874,87.106,19.726,-178.6245,-1.1234,0.0000
C01835=49.917,85.194,19.692,-177.1700,-3.1394,0.0000
C01836=51.163,83.502,19.627,-176.4596,-6.1367,0.0000
C01837=51.961,81.931,19.493,-175.4388,-10.0982,0.0000
C01838=52.755,80.388,19.309,-171.7459,-14.7954,0.0000
C01839=53.950,78.738,19.120,-165.3859,-17.8376,0.0000
C01840=56.048,76.685,18.976,-160.0061,-17.9537,0.0000
C01841=59.448,73.859,18.917,-158.5554,-18.0210,0.0000
C01842=63.169,70.689,18.914,-159.1041,-18.7952,0.0000
C01843=67.036,67.036,18.916,-160.1239,-19.8761,0.0000
C01844=70.689,63.169,18.914,-161.2048,-20.8959,0.0000
C01845=73.859,59.448,18.917,-161.9790,-21.4446,0.0000
C01846=76.685,56.048,18.976,-162.0463,-19.9939,0.0000
C01847=78.738,53.950,19.120,-162.1624,-14.6141,0.0000
C01848=80.388,52.755,19.309,-165.2046,-8.2541,0.0000
C01849=81.931,51.961,19.493,-169.9018,-4.5612,0.0000
C01850=83.502,51.163,19.627,-173.8633,-3.5404,0.0000
C01851=85.194,49.917,19.692,-176.8606,-2.8300,0.0000
C01852=87.106,47.874,19.726,-178.8766,-1.3755,0.0000
C01853=88.975,45.272,19.753,-179.8510,-0.2292,0.0000
C01854=90.515,42.449,19.780,-179.9656,-0.0688,0.0000
C01855=91.796,39.659,19.798,-179.9943,-0.0057,0.0000
C01856=92.953,36.867,19.798,-179.9943,-0.0057,0.0000
C01857=94.020,33.988,19.780,-179.9771,-0.0745,0.0000
C01858=94.927,30.903,19.753,-179.9370,-0.2693,0.0000
C01859=95.446,27.741,19.726,-179.8223,-1.7650,0.0000
C01860=95.538,24.945,19.692,179.7817,-4.2207,0.0000
C01861=95.222,22.867,19.627,178.1531,-6.8321,0.0000
C01862=94.676,21.192,19.493,176.0252,-10.3357,0.0000
C01863=94.146,19.540,19.309,175.1883,-16.1404,0.0000
C01864=93.824,17.528,19.120,177.5271,-22.3839,0.0000
C01865=93.857,14.592,18.976,-178.3880,-25.9396,0.0000
C01866=94.262,10.190,18.917,-177.2685,-26.9190,0.0000
C01867=94.652,5.317,18.914,-178.3272,-27.0495,0.0000
C01868=94.804,0.000,18.916,180.0000,-27.0775,0.0000
C01869=94.652,-5.317,18.914,178.3272,-27.0495,0.0000
C01870=94.262,-10.190,18.917,177.2685,-26.9190,0.0000
C01871=93.857,-14.592,18.976,178.3880,-25.9396,0.0000
C01872=93.824,-17.528,19.120,-177.5271,-22.3839,0.0000
C01873=94.146,-19.540,19.309,-175.1883,-16.1404,0.0000
C01874=94.676,-21.192,19.493,-176.0252,-10.3357,0.0000
C01875=95.222,-22.867,19.627,-178.1531,-6.8321,0.0000
C01876=95.538,-24.945,19.692,-179.7817,-4.2207,0.0000
C01877=95.446,-27.741,19.726,179.8223,-1.7650,0.0000
C01878=94.927,-30.903,19.753,179.9370,-0.2693,0.0000
C01879=94.020,-33.988,19.780,179.9771,-0.0745,0.0000
C01880=92.953,-36.867,19.798,179.9943,-0.0057,0.0000
C01881=91.796,-39.659,19.798,179.9943,-0.0057,0.0000
C01882=90.515,-42.449,19.780,179.9656,-0.0688,0.0000
C01883=88.975,-45.272,19.753,179.8510,-0.2292,0.0000
C01884=87.106,-47.874,19.726,178.8766,-1.3755,0.0000
C01885=85.194,-49.917,19.692,176.8606,-2.8300,0.0000
C01886=83.502,-51.163,19.627,173.8633,-3.5404,0.0000
C01887=81.931,-51.961,19.493,169.9018,-4.5612,0.0000
C01888=80.388,-52.755,19.309,165.2046,-8.2541,0.0000
C01889=78.738,-53.950,19.120,162.1624,-14.6141,0.0000
C01890=76.685,-56.048,18.976,162.0463,-19.9939,0.0000
C01891=73.859,-59.448,18.917,161.9790,-21.4446,0.0000
C01892=70.689,-63.169,18.914,161.2048,-20.8959,0.0000
